   REGION FB Scanner
       #sScannerComm(iInit := "LBP_Chan1".A_Ref,
                     iReady := "DB_OPC_Laser".Scanner.In.Ready,
                     iStatus := "DB_OPC_Laser".Scanner.In.Status,
                     iStatusDescription := "DB_OPC_Laser".Scanner.In.StatusDescription,
                     iCheckNumber := "DB_OPC_Laser".Scanner.In.CheckNumber,
                     iPartOnFixture := "DB_PartManagement".sPosition.sFixture.Undrilled.Presence.Part OR "DB_PartManagement".sPosition.sFixture.Drilled.Presence.Part,
                     iStationNumber := #sScannerComm.iStationNumber,
                     iHoleNumber := #sScannerComm.iHoleNumber,
                     iJobListName := #sScannerComm.iJobListName,
                     iJobName := #sScannerComm.iJobName,
                     iMeasureZ := #sMeasureZ,
                     oEndOfJob => #sScannerComm.oEndOfJob,
                     ioRequestJob := "DB_OPC_Laser".Scanner.Out.RequestJob,
                     ioCheckNumber := "DB_OPC_Laser".Scanner.Out.CheckNumber,
                     oIsFirstJobOfPiece => "DB_OPC_Laser".Scanner.Out.Parameters.IsFirstJobOfPiece,
                     oStationNumber => "DB_OPC_Laser".Scanner.Out.Parameters.StationNumber,
                     oHoleNumber => "DB_OPC_Laser".Scanner.Out.Parameters.HoleNumber,
                     oJobListName => "DB_OPC_Laser".Scanner.Out.Parameters.JobListName,
                     oJobName => "DB_OPC_Laser".Scanner.Out.Parameters.JobName,
                     oMeasureZ => "DB_OPC_Laser".Scanner.Out.Parameters.MeasureZ,
                     oBadPart => #sScannerComm.oBadPart,
                     oGoodPart => #sScannerComm.oGoodPart,
                     ioRequestJob_NC := #sScannerComm.ioRequestJob_NC,
                     ioReady_NC := #sScannerComm.ioReady_NC);
   END_REGION

   REGION End of Job
       #sTimePulseWriteParam(IN := #sWriteR_ParamReq,
                             PT := T#100ms);
       IF #sTimePulseWriteParam.Q THEN
           #sWriteR_ParamReq := FALSE;
       END_IF;


       IF #sScannerComm.oEndOfJob THEN
           #sR96 := 0;
           #sR97 := 1;
           #sWriteR_ParamReq := TRUE;
       END_IF;

       IF #sWriteR_Param.Done THEN
           #sWriteR_ParamReq := FALSE;
       END_IF;
   END_REGION
END_FUNCTION_BLOCK

FUNCTION_BLOCK "FB_ScannerComm"   // FB85, SCL
{ S7_Optimized_Access := 'TRUE' }
// stored: MemoryReserve 100, SetENOAutomatically false
   VAR_INPUT
      iInit : Bool;
      iReady : Bool;   // From HMI OPC UA
      iStatus : DInt;   // From HMI OPC UA
      iStatusDescription : String;   // From HMI OPC UA
      iCheckNumber : Byte;   // From HMI OPC UA
      iPartOnFixture : Bool;
      iStationNumber : Byte;   // From NC ?
      iHoleNumber : DInt;   // From NC ?
      iJobListName : String;   // From NC ?
      iJobName : DInt;   // From NC ?
      iMeasureZ : LReal;   // From NC ?
   END_VAR
   VAR_OUTPUT
      oIsFirstJobOfPiece : Bool;
      oStationNumber : Byte;
      oHoleNumber : DInt;
      oJobListName : String;
      oJobName : String;
      oMeasureZ : LReal;
      oBadPart : Bool;
      oGoodPart : Bool;
      oEndOfJob : Bool;
   END_VAR
   VAR_IN_OUT
      ioRequestJob_NC : Bool;   // From NC ?
      ioReady_NC : Bool;   // From NC ?
      ioCheckNumber : Byte;
      ioRequestJob : Bool;
   END_VAR
   VAR
      sRT_PartOnFixture : R_TRIG;
      sRT_Ready { S7_SetPoint := 'True'} : R_TRIG;
      sEndOfJob { S7_SetPoint := 'True'} : Bool;
      sRT_RequestJob_NC : R_TRIG;
      sJobListName { S7_SetPoint := 'True'} : String;
      sJobName : String;
      sJobInProgress : Bool;
   END_VAR
BEGIN
   REGION Description header 
       //==================================================================================
       // POSALUX Swiss SA / (C) Copyright 2026
       //----------------------------------------------------------------------------------
       // Title: FB_ScannerComm
       // Comment/Function: 
       //
       // Author: Fabien WALDT
       // Engineering: TIA Portal v20
       //----------------------------------------------------------------------------------
       // Change log table:
       // Version  | Date     | Expert in charge | Changes applied
       // ---------|----------|------------------|------------------------------------
       // 00.00.01 | 20260330 | WFA              | First released version
       // ==================================================================================
   END_REGION

   REGION R_Trig
       #sRT_PartOnFixture(CLK := #iPartOnFixture);

       #sRT_Ready(CLK := #iReady);
       #sEndOfJob := #sRT_Ready.Q AND #sJobInProgress;

       #sRT_RequestJob_NC(CLK := #ioRequestJob_NC);
   END_REGION

   REGION Job
   #sJobListName := #iJobListName;
   #sJobName := DINT_TO_STRING(IN := #iJobName);

   IF #sJobName[1] = '+' THEN
       #sJobName := DELETE(IN := #sJobName, L := 1, P := 1);
   END_IF;
   END_REGION

   REGION Parameters
       // IsFirstJobOfPiece 
       IF #sRT_PartOnFixture.Q THEN
           #oIsFirstJobOfPiece := TRUE;
       ELSIF #sEndOfJob OR NOT #iPartOnFixture THEN
           #oIsFirstJobOfPiece := FALSE;
       END_IF;

       IF #sRT_RequestJob_NC.Q THEN
           // StationNumber 
           #oStationNumber := #iStationNumber;

           // HoleNumber 
           #oHoleNumber := #iHoleNumber;

           // JobListName 
           #oJobListName := #sJobListName;

           // JobName 
           #oJobName := #sJobName;

           // MeasureZ 
           #oMeasureZ := #iMeasureZ;

           // CheckNumber Increment
           #ioCheckNumber := #ioCheckNumber + 1;
           IF #ioCheckNumber > 255 OR #ioCheckNumber < 1 THEN
               #ioCheckNumber := 1;
           END_IF;

           // Reset Bad/Good Part
           #oBadPart := FALSE;
           #oGoodPart := FALSE;
       END_IF;
   END_REGION

   REGION Request Job
       IF #ioRequestJob_NC AND #iReady AND NOT #sJobInProgress THEN
           #sJobInProgress := TRUE;
           #ioRequestJob := TRUE;
       ELSIF (#ioRequestJob AND NOT #iReady) OR #iInit THEN
           #ioRequestJob := FALSE;
       END_IF;
   END_REGION

   REGION End of Job
       IF #sEndOfJob THEN
           IF #ioCheckNumber = #iCheckNumber AND #iStatus = 1 THEN
               #oGoodPart := TRUE;
           ELSE
               #oBadPart := TRUE;
           END_IF;
           #sJobInProgress := FALSE;
       END_IF;

       // Update Output
       #oEndOfJob := #sEndOfJob;
   END_REGION
END_FUNCTION_BLOCK

FUNCTION_BLOCK "FB_Part_Data"   // FB93, SCL
{ S7_Optimized_Access := 'TRUE' }
// stored: MemoryReserve 100, SetENOAutomatically false
   VAR
      Part_Data_Ident : "FB_ReadWrite_GUDs";
      sWriteDataEnable { S7_SetPoint := 'True'} : Bool;
      sNewPartDataIdent : Bool;
      RT_NewPartDataIdent : R_TRIG;
      sCurrentPartDataIdent { S7_SetPoint := 'True'} : String;
   END_VAR
   VAR_TEMP
      tIndex : Int;
   END_VAR
BEGIN
   REGION Description header 
       //==================================================================================
       // POSALUX Swiss SA / (C) Copyright 2026
       //----------------------------------------------------------------------------------
       // Title: FB_Part_Data
       // Comment/Function: 
       //
       // Author: Fabien WALDT
       // Engineering: TIA Portal v20
       //----------------------------------------------------------------------------------
       // Change log table:
       // Version  | Date     | Expert in charge | Changes applied
       // ---------|----------|------------------|------------------------------------
       // 00.00.01 | 20260518 | WFA              | First released version
       // ==================================================================================
   END_REGION

   REGION Data Init
       #Part_Data_Ident.sName := 'PART_DATA_IDENT';
       #Part_Data_Ident.sType := 4;
       #Part_Data_Ident.sNCK_channel := 1;
    //   #Part_Data_Ident.sWriteVal_String[0] := 'Test_ID_From_PLC';
   END_REGION

   REGION Call Read/Wrtite GUD
       #Part_Data_Ident();
   END_REGION

   REGION Convert DMC into String

   END_REGION

   REGION New Value
   // Convert DMC Array into String    
   Chars_TO_Strg(Chars:= "DB_DataPositions".Position[4].DMC,
                 pChars:= 0,
                 Cnt:= 19,
                 Strg=> #sCurrentPartDataIdent);

   // Check if new Part on Fixture
   IF #Part_Data_Ident.sWriteVal_String[0] <> #sCurrentPartDataIdent THEN
       #Part_Data_Ident.sWriteVal_String[0] := #sCurrentPartDataIdent;
       #sNewPartDataIdent := TRUE;
       END_IF;
   END_REGION

   // Il faut tout d'abord effectuer une lecture :
   // #Part_Data_Ident.sStart_rd
   // Pour obtenir #Part_Data_Ident.sRead_done
   // On peut alors effctuer une ecriture avec #Part_Data_Ident.sStart_wr
   // Pour obtenir #Part_Data_Ident.sWrite_done

   REGION Write Datas Request
       IF NOT #sWriteDataEnable THEN
           #Part_Data_Ident.sStart_rd := TRUE;
       END_IF;

   IF #Part_Data_Ident.sRead_done THEN
       #Part_Data_Ident.sStart_rd := FALSE;
       #sWriteDataEnable := TRUE;
   END_IF;

   #RT_NewPartDataIdent(CLK := #sNewPartDataIdent);
   IF #RT_NewPartDataIdent.Q AND #sWriteDataEnable THEN
       #Part_Data_Ident.sStart_wr := TRUE;
       #sNewPartDataIdent := FALSE;
   ELSIF #Part_Data_Ident.sWrite_done THEN
       #Part_Data_Ident.sStart_wr := FALSE;
   END_IF;
   END_REGION
END_FUNCTION_BLOCK

FUNCTION_BLOCK "FB_ReadWrite_GUDs"   // FB1200, SCL
{ S7_Optimized_Access := 'TRUE' }
// stored: AutoNumber false, MemoryReserve 100, SetENOAutomatically false
   VAR
      sStart_rd { ExternalAccessible := 'False'; ExternalVisible := 'False'; ExternalWritable := 'False'} : Bool;
      sNCK_channel { ExternalAccessible := 'False'; ExternalVisible := 'False'; ExternalWritable := 'False'} : Byte;   // 0:GUD NCK, 1:GUD Chan1, 2:GUD Chan2 etc...
      sType { ExternalAccessible := 'False'; ExternalVisible := 'False'; ExternalWritable := 'False'} : Int;   // 0:Bool, 1:Int, 2:DWord, 3:Real, 4:String
      sName { ExternalAccessible := 'False'; ExternalVisible := 'False'; ExternalWritable := 'False'} : String;   // GUD Name
      sIndex1 { ExternalAccessible := 'False'; ExternalVisible := 'False'; ExternalWritable := 'False'} : Int;
      sindex2 { ExternalAccessible := 'False'; ExternalVisible := 'False'; ExternalWritable := 'False'} : Int;
      sToken_GUD { ExternalAccessible := 'False'; ExternalVisible := 'False'; ExternalWritable := 'False'} : "UDT_Token_GUD";
      sValue_bit { ExternalAccessible := 'False'; ExternalVisible := 'False'; ExternalWritable := 'False'} : Bool;
      sValue_int { ExternalAccessible := 'False'; ExternalVisible := 'False'; ExternalWritable := 'False'} : Int;
      sValue_double { ExternalAccessible := 'False'; ExternalVisible := 'False'; ExternalWritable := 'False'} : DWord;
      sValue_real { ExternalAccessible := 'False'; ExternalVisible := 'False'; ExternalWritable := 'False'} : Real;
      sValue_String { ExternalAccessible := 'False'; ExternalVisible := 'False'; ExternalWritable := 'False'} : String;
      sStatus_rd { ExternalAccessible := 'False'; ExternalVisible := 'False'; ExternalWritable := 'False'} : Word;
      sRead_done { ExternalAccessible := 'False'; ExternalVisible := 'False'; ExternalWritable := 'False'} : Bool;
      sRead_done_Mem { ExternalAccessible := 'False'; ExternalVisible := 'False'; ExternalWritable := 'False'} : Bool;
      sStart_wr { ExternalAccessible := 'False'; ExternalVisible := 'False'; ExternalWritable := 'False'} : Bool;
      sNumVar_wr { ExternalAccessible := 'False'; ExternalVisible := 'False'; ExternalWritable := 'False'} : Int := 1;
      sAddr_wr { ExternalAccessible := 'False'; ExternalVisible := 'False'; ExternalWritable := 'False'} : Array[0..7] of "UDT_Token_GUD";
      sColumn_wr { ExternalAccessible := 'False'; ExternalVisible := 'False'; ExternalWritable := 'False'} : Array[0..7] of Word;
      sLine_wr { ExternalAccessible := 'False'; ExternalVisible := 'False'; ExternalWritable := 'False'} : Array[0..7] of Word;
      sStatus_wr { ExternalAccessible := 'False'; ExternalVisible := 'False'; ExternalWritable := 'False'} : Word;
      sWrite_done { ExternalAccessible := 'False'; ExternalVisible := 'False'; ExternalWritable := 'False'} : Bool;
      sWriteVal_bit { ExternalAccessible := 'False'; ExternalVisible := 'False'; ExternalWritable := 'False'} : Array[0..7] of Bool;
      sWriteVal_int { ExternalAccessible := 'False'; ExternalVisible := 'False'; ExternalWritable := 'False'} : Array[0..7] of Int;
      sWriteVal_double { ExternalAccessible := 'False'; ExternalVisible := 'False'; ExternalWritable := 'False'} : Array[0..7] of DWord;
      sWriteVal_Real { ExternalAccessible := 'False'; ExternalVisible := 'False'; ExternalWritable := 'False'} : Array[0..7] of DWord;
      sWriteVal_String { ExternalAccessible := 'False'; ExternalVisible := 'False'; ExternalWritable := 'False'} : Array[0..7] of String;
      sLBP_ReadGUD_Instance { ExternalAccessible := 'False'; ExternalVisible := 'False'; ExternalWritable := 'False'} : "LBP_ReadGUD";
      sLBP_WriteGUD_Instance { ExternalAccessible := 'False'; ExternalVisible := 'False'; ExternalWritable := 'False'} : "LBP_WriteVar";
   END_VAR
   VAR_TEMP
      tArea : Byte;
      tUnit : Byte;
      tError : Bool;
      tStatus : Word;
      tLoop_I : Int;
   END_VAR
   // sColumn_wr[0..7] := 16#1;
   // sLine_wr[0..7] := 16#1;
BEGIN
   REGION Reading
       IF #sNCK_channel = 0 THEN
           #tArea := 0;
           #tUnit := 1;
       ELSE
           #tArea := 2;
           #tUnit := #sNCK_channel;
       END_IF;

       CASE #sType OF
           0:
               #sLBP_ReadGUD_Instance(Req := #sStart_rd,
                                     Addr := #sName,
                                     Area := #tArea,
                                     Unit := #tUnit,
                                     Index1 := #sIndex1,
                                     Index2 := #sindex2,
                                     CnvtToken := TRUE,
                                     VarToken := #sToken_GUD,
                                     Error => #tError,
                                     Done => #sRead_done,
                                     State => #tStatus,
                                     RD := #sValue_bit);
           1:
               #sLBP_ReadGUD_Instance(Req := #sStart_rd,
                                     Addr := #sName,
                                     Area := #tArea,
                                     Unit := #tUnit,
                                     Index1 := #sIndex1,
                                     Index2 := #sindex2,
                                     CnvtToken := TRUE,
                                     VarToken := #sToken_GUD,
                                     Error => #tError,
                                     Done => #sRead_done,
                                     State => #tStatus,
                                     RD := #sValue_int);

           2:
               #sLBP_ReadGUD_Instance(Req := #sStart_rd,
                                     Addr := #sName,
                                     Area := #tArea,
                                     Unit := #tUnit,
                                     Index1 := #sIndex1,
                                     Index2 := #sindex2,
                                     CnvtToken := TRUE,
                                     VarToken := #sToken_GUD,
                                     Error => #tError,
                                     Done => #sRead_done,
                                     State => #tStatus,
                                     RD := #sValue_double);

           3:
               #sLBP_ReadGUD_Instance(Req := #sStart_rd,
                                     Addr := #sName,
                                     Area := #tArea,
                                     Unit := #tUnit,
                                     Index1 := #sIndex1,
                                     Index2 := #sindex2,
                                     CnvtToken := TRUE,
                                     VarToken := #sToken_GUD,
                                     Error => #tError,
                                     Done => #sRead_done,
                                     State => #tStatus,
                                     RD := #sValue_real);

           4:
               #sLBP_ReadGUD_Instance(Req := #sStart_rd,
                                     Addr := #sName,
                                     Area := #tArea,
                                     Unit := #tUnit,
                                     Index1 := #sIndex1,
                                     Index2 := #sindex2,
                                     CnvtToken := TRUE,
                                     VarToken := #sToken_GUD,
                                     Error => #tError,
                                     Done => #sRead_done,
                                     State => #tStatus,
                                     RD := #sValue_String);


       END_CASE;

       IF #sRead_done OR #tError THEN
           #sRead_done := TRUE;
           #sStatus_rd := #tStatus;
           #sStart_rd := FALSE;
       END_IF;
       IF #sRead_done AND NOT #sRead_done_Mem THEN
           FOR #tLoop_I := 1 TO 8 DO
               IF #tLoop_I <= #sNumVar_wr THEN
                 #sAddr_wr[#tLoop_I - 1] := #sToken_GUD;
               END_IF;
           END_FOR;
           #sRead_done_Mem := TRUE;
       END_IF;

   END_REGION


   REGION Writing

       CASE #sType OF
           0:
               #sLBP_WriteGUD_Instance(Req := #sStart_wr AND #sRead_done_Mem,
                                      NumVar := #sNumVar_wr,
                                      Addr1 := #sAddr_wr[0],
                                      Line1 := #sLine_wr[0],
                                      Column1 := #sColumn_wr[0],
                                      Addr2 := #sAddr_wr[1],
                                      Line2 := #sLine_wr[1],
                                      Column2 := #sColumn_wr[1],
                                      Addr3 := #sAddr_wr[2],
                                      Line3 := #sLine_wr[2],
                                      Column3 := #sColumn_wr[2],
                                      Addr4 := #sAddr_wr[3],
                                      Line4 := #sLine_wr[3],
                                      Column4 := #sColumn_wr[3],
                                      Addr5 := #sAddr_wr[4],
                                      Line5 := #sLine_wr[4],
                                      Column5 := #sColumn_wr[4],
                                      Addr6 := #sAddr_wr[5],
                                      Line6 := #sLine_wr[5],
                                      Column6 := #sColumn_wr[5],
                                      Addr7 := #sAddr_wr[6],
                                      Line7 := #sLine_wr[6],
                                      Column7 := #sColumn_wr[6],
                                      Addr8 := #sAddr_wr[7],
                                      Line8 := #sLine_wr[7],
                                      Column8 := #sColumn_wr[7],
                                      Error => #tError,
                                      Done => #sWrite_done,
                                      State => #tStatus,
                                      SD1 := #sWriteVal_bit[0],
                                      SD2 := #sWriteVal_bit[1],
                                      SD3 := #sWriteVal_bit[2],
                                      SD4 := #sWriteVal_bit[3],
                                      SD5 := #sWriteVal_bit[4],
                                      SD6 := #sWriteVal_bit[5],
                                      SD7 := #sWriteVal_bit[6],
                                      SD8 := #sWriteVal_bit[7]);
           1:
               #sLBP_WriteGUD_Instance(Req := #sStart_wr AND #sRead_done_Mem,
                                      NumVar := #sNumVar_wr,
                                      Addr1 := #sAddr_wr[0],
                                      Line1 := #sLine_wr[0],
                                      Column1 := #sColumn_wr[0],
                                      Addr2 := #sAddr_wr[1],
                                      Line2 := #sLine_wr[1],
                                      Column2 := #sColumn_wr[1],
                                      Addr3 := #sAddr_wr[2],
                                      Line3 := #sLine_wr[2],
                                      Column3 := #sColumn_wr[2],
                                      Addr4 := #sAddr_wr[3],
                                      Line4 := #sLine_wr[3],
                                      Column4 := #sColumn_wr[3],
                                      Addr5 := #sAddr_wr[4],
                                      Line5 := #sLine_wr[4],
                                      Column5 := #sColumn_wr[4],
                                      Addr6 := #sAddr_wr[5],
                                      Line6 := #sLine_wr[5],
                                      Column6 := #sColumn_wr[5],
                                      Addr7 := #sAddr_wr[6],
                                      Line7 := #sLine_wr[6],
                                      Column7 := #sColumn_wr[6],
                                      Addr8 := #sAddr_wr[7],
                                      Line8 := #sLine_wr[7],
                                      Column8 := #sColumn_wr[7],
                                      Error => #tError,
                                      Done => #sWrite_done,
                                      State => #tStatus,
                                      SD1 := #sWriteVal_int[0],
                                      SD2 := #sWriteVal_int[1],
                                      SD3 := #sWriteVal_int[2],
                                      SD4 := #sWriteVal_int[3],
                                      SD5 := #sWriteVal_int[4],
                                      SD6 := #sWriteVal_int[5],
                                      SD7 := #sWriteVal_int[6],
                                      SD8 := #sWriteVal_int[7]);

           2:
               #sLBP_WriteGUD_Instance(Req := #sStart_wr AND #sRead_done_Mem,
                                      NumVar := #sNumVar_wr,
                                      Addr1 := #sAddr_wr[0],
                                      Line1 := #sLine_wr[0],
                                      Column1 := #sColumn_wr[0],
                                      Addr2 := #sAddr_wr[1],
                                      Line2 := #sLine_wr[1],
                                      Column2 := #sColumn_wr[1],
                                      Addr3 := #sAddr_wr[2],
                                      Line3 := #sLine_wr[2],
                                      Column3 := #sColumn_wr[2],
                                      Addr4 := #sAddr_wr[3],
                                      Line4 := #sLine_wr[3],
                                      Column4 := #sColumn_wr[3],
                                      Addr5 := #sAddr_wr[4],
                                      Line5 := #sLine_wr[4],
                                      Column5 := #sColumn_wr[4],
                                      Addr6 := #sAddr_wr[5],
                                      Line6 := #sLine_wr[5],
                                      Column6 := #sColumn_wr[5],
                                      Addr7 := #sAddr_wr[6],
                                      Line7 := #sLine_wr[6],
                                      Column7 := #sColumn_wr[6],
                                      Addr8 := #sAddr_wr[7],
                                      Line8 := #sLine_wr[7],
                                      Column8 := #sColumn_wr[7],
                                      Error => #tError,
                                      Done => #sWrite_done,
                                      State => #tStatus,
                                      SD1 := #sWriteVal_double[0],
                                      SD2 := #sWriteVal_double[1],
                                      SD3 := #sWriteVal_double[2],
                                      SD4 := #sWriteVal_double[3],
                                      SD5 := #sWriteVal_double[4],
                                      SD6 := #sWriteVal_double[5],
                                      SD7 := #sWriteVal_double[6],
                                      SD8 := #sWriteVal_double[7]);

           3:
               #sLBP_WriteGUD_Instance(Req := #sStart_wr AND #sRead_done_Mem,
                                      NumVar := #sNumVar_wr,
                                      Addr1 := #sAddr_wr[0],
                                      Line1 := #sLine_wr[0],
                                      Column1 := #sColumn_wr[0],
                                      Addr2 := #sAddr_wr[1],
                                      Line2 := #sLine_wr[1],
                                      Column2 := #sColumn_wr[1],
                                      Addr3 := #sAddr_wr[2],
                                      Line3 := #sLine_wr[2],
                                      Column3 := #sColumn_wr[2],
                                      Addr4 := #sAddr_wr[3],
                                      Line4 := #sLine_wr[3],
                                      Column4 := #sColumn_wr[3],
                                      Addr5 := #sAddr_wr[4],
                                      Line5 := #sLine_wr[4],
                                      Column5 := #sColumn_wr[4],
                                      Addr6 := #sAddr_wr[5],
                                      Line6 := #sLine_wr[5],
                                      Column6 := #sColumn_wr[5],
                                      Addr7 := #sAddr_wr[6],
                                      Line7 := #sLine_wr[6],
                                      Column7 := #sColumn_wr[6],
                                      Addr8 := #sAddr_wr[7],
                                      Line8 := #sLine_wr[7],
                                      Column8 := #sColumn_wr[7],
                                      Error => #tError,
                                      Done => #sWrite_done,
                                      State => #tStatus,
                                      SD1 := #sWriteVal_Real[0],
                                      SD2 := #sWriteVal_Real[1],
                                      SD3 := #sWriteVal_Real[2],
                                      SD4 := #sWriteVal_Real[3],
                                      SD5 := #sWriteVal_Real[4],
                                      SD6 := #sWriteVal_Real[5],
                                      SD7 := #sWriteVal_Real[6],
                                      SD8 := #sWriteVal_Real[7]);

           4:
               #sLBP_WriteGUD_Instance(Req := #sStart_wr AND #sRead_done_Mem,
                                      NumVar := #sNumVar_wr,
                                      Addr1 := #sAddr_wr[0],
                                      Line1 := #sLine_wr[0],
                                      Column1 := #sColumn_wr[0],
                                      Addr2 := #sAddr_wr[1],
                                      Line2 := #sLine_wr[1],
                                      Column2 := #sColumn_wr[1],
                                      Addr3 := #sAddr_wr[2],
                                      Line3 := #sLine_wr[2],
                                      Column3 := #sColumn_wr[2],
                                      Addr4 := #sAddr_wr[3],
                                      Line4 := #sLine_wr[3],
                                      Column4 := #sColumn_wr[3],
                                      Addr5 := #sAddr_wr[4],
                                      Line5 := #sLine_wr[4],
                                      Column5 := #sColumn_wr[4],
                                      Addr6 := #sAddr_wr[5],
                                      Line6 := #sLine_wr[5],
                                      Column6 := #sColumn_wr[5],
                                      Addr7 := #sAddr_wr[6],
                                      Line7 := #sLine_wr[6],
                                      Column7 := #sColumn_wr[6],
                                      Addr8 := #sAddr_wr[7],
                                      Line8 := #sLine_wr[7],
                                      Column8 := #sColumn_wr[7],
                                      Error => #tError,
                                      Done => #sWrite_done,
                                      State => #tStatus,
                                      SD1 := #sWriteVal_String[0],
                                      SD2 := #sWriteVal_String[1],
                                      SD3 := #sWriteVal_String[2],
                                      SD4 := #sWriteVal_String[3],
                                      SD5 := #sWriteVal_String[4],
                                      SD6 := #sWriteVal_String[5],
                                      SD7 := #sWriteVal_String[6],
                                      SD8 := #sWriteVal_String[7]);
       END_CASE;

       IF #sWrite_done OR #tError THEN
           #sWrite_done := TRUE;
           #sStatus_wr := #tStatus;
           #sStart_wr := FALSE;
       END_IF;


   END_REGION
END_FUNCTION_BLOCK

FUNCTION_BLOCK "FB_Recipe"   // FB81, SCL
{ S7_Optimized_Access := 'TRUE' }
// stored: AutoNumber false, MemoryReserve 100, SetENOAutomatically false
BEGIN
   REGION Description header 
       //==================================================================================
       // POSALUX Swiss SA / (C) Copyright 2026
       //----------------------------------------------------------------------------------
       // Title: FB_Recipe
       // Comment/Function: 
       //
       // Author: Fabien WALDT
       // Engineering: TIA Portal v20
       //----------------------------------------------------------------------------------
       // Change log table:
       // Version  | Date     | Expert in charge | Changes applied
       // ---------|----------|------------------|------------------------------------
       // 00.00.01 | 20260427 | WFA              | First released version
       // ==================================================================================
   END_REGION

   REGION Current
       "DB_OPC_Recipe".Current.RecipeId := "DB_OPC_Recipe".Current.RecipeId;
       "DB_OPC_Recipe".Current.RecipeVersionGuid := "DB_OPC_Recipe".Current.RecipeVersionGuid;
   END_REGION

   REGION Data
       "DB_OPC_Recipe".Data.LaserJobListName := "DB_OPC_Recipe".Data.LaserJobListName;
       "DB_OPC_Recipe".Data.RecipeId := "DB_OPC_Recipe".Data.RecipeId;
       "DB_OPC_Recipe".Data.RecipeName := "DB_OPC_Recipe".Data.RecipeName;
       "DB_OPC_Recipe".Data.RecipeVersionGuid := "DB_OPC_Recipe".Data.RecipeVersionGuid;

       // Station 1
       // General \ Detections \ WorkPart
       "DB_OPC_Recipe".Data.Station1.General.Detections.WorkPart.Max := "DB_OPC_Recipe".Data.Station1.General.Detections.WorkPart.Max;
       "DB_OPC_Recipe".Data.Station1.General.Detections.WorkPart.Min := "DB_OPC_Recipe".Data.Station1.General.Detections.WorkPart.Min;
       // General \ GasPressure
        "DB_OPC_Recipe".Data.Station1.General.GazPressure.WorkLaserDefault := "DB_OPC_Recipe".Data.Station1.General.GazPressure.WorkLaserDefault;
   END_REGION

   REGION TransfertToPlc
       IF "DB_OPC_Recipe".TransferToPlc THEN
           "DB_OPC_Recipe".Current.RecipeId := "DB_OPC_Recipe".Data.RecipeId;
           "DB_OPC_Recipe".Current.RecipeVersionGuid := "DB_OPC_Recipe".Data.RecipeVersionGuid;
           "DB_Scanner".sScannerComm.iJobListName := "DB_OPC_Recipe".Data.LaserJobListName;
       //    "DB_HMISetting".GasAssistSetPoint := LREAL_TO_REAL("DB_OPC_Recipe".Data.Station1.General.GazPressure.WorkLaserDefault);   WAF A LIBERER QUAND RECETTE OK
       //    "DB_GestionFixture".sFixturePartControl.iProdOK_LimHigh := LREAL_TO_REAL("DB_OPC_Recipe".Data.Station1.General.Detections.WorkPart.Max);  WAF A LIBERER QUAND RECETTE OK
       //    "DB_GestionFixture".sFixturePartControl.iProdOK_LimLow := LREAL_TO_REAL("DB_OPC_Recipe".Data.Station1.General.Detections.WorkPart.Min);   WAF A LIBERER QUAND RECETTE OK
           "DB_OPC_Recipe".TransferToPlc := FALSE;
       END_IF;
   END_REGION
END_FUNCTION_BLOCK

FUNCTION_BLOCK "FB_PartManagement"   // FB86, SCL
{ S7_Optimized_Access := 'TRUE' }
// stored: MemoryReserve 100, SetENOAutomatically false
   VAR
      sShuttle1DrilledPart : "FB_StatusPart";
      sShuttle1UndrilledPart { S7_SetPoint := 'True'} : "FB_StatusPart";
      sShuttle2DrilledPart { S7_SetPoint := 'True'} : "FB_StatusPart";
      sShuttle2UndrilledPart { S7_SetPoint := 'True'} : "FB_StatusPart";
      sShuttle1DrilledBw : "FB_StatusPart";
      sShuttle1UndrilledBw { S7_SetPoint := 'True'} : "FB_StatusPart";
      sShuttle2DrilledBw { S7_SetPoint := 'True'} : "FB_StatusPart";
      sShuttle2UndrilledBw { S7_SetPoint := 'True'} : "FB_StatusPart";
      sGripperDrilledPart : "FB_StatusPart";
      sGripperUndrilledPart { S7_SetPoint := 'True'} : "FB_StatusPart";
      sGripperDrilledBw : "FB_StatusPart";
      sGripperUndrilledBw { S7_SetPoint := 'True'} : "FB_StatusPart";
      sFixtureDrilledPart : "FB_StatusPart";
      sFixtureUndrilledPart { S7_SetPoint := 'True'} : "FB_StatusPart";
      sFixtureDrilledBw : "FB_StatusPart";
      sFixtureUndrilledBw { S7_SetPoint := 'True'} : "FB_StatusPart";
      sPosition { S7_SetPoint := 'True'} : "FB_Position";
   END_VAR
BEGIN
   REGION Description header 
       //==================================================================================
       // POSALUX Swiss SA / (C) Copyright 2026
       //----------------------------------------------------------------------------------
       // Title: FB_PartManagement
       // Comment/Function: 
       //
       // Author: Fabien WALDT
       // Engineering: TIA Portal v20
       //----------------------------------------------------------------------------------
       // Change log table:
       // Version  | Date     | Expert in charge | Changes applied
       // ---------|----------|------------------|------------------------------------
       // 00.00.01 | 20260310 | WFA              | First released version
       // ==================================================================================
   END_REGION

   REGION Shuttle 1 States
       // Drilled Part
       #sShuttle1DrilledPart(iGood := #sPosition.sShuttle1.Drilled.Presence.Part AND NOT #sShuttle1DrilledPart.iBad,
                             iUnknown := #sShuttle1DrilledPart.iUnknown,
                             iBad := #sShuttle1DrilledPart.iBad,
                             iAbsent := NOT #sPosition.sShuttle1.Drilled.Presence.Part,
                             iPresentUnexpected := "DB_LoaderShuttle1".sControlIn.sExtraPartCtrlDrilled OR "DB_LoaderShuttle1".sControlOut.sExtraPartCtrlDrilled,
                             iAbsentUnexpected := "DB_LoaderShuttle1".sControlIn.sMissingPartCtrlDrilled OR "DB_LoaderShuttle1".sControlOut.sMissingPartCtrlDrilled,
                             oStatus => #sPosition.sShuttle1.Drilled.States.Part);

       // Undrilled Part
       #sShuttle1UndrilledPart(iGood := #sPosition.sShuttle1.Undrilled.Presence.Part AND NOT #sShuttle1UndrilledPart.iBad,
                               iUnknown := #sShuttle1UndrilledPart.iUnknown,
                               iBad := #sShuttle1UndrilledPart.iBad,
                               iAbsent := NOT #sPosition.sShuttle1.Undrilled.Presence.Part,
                               iPresentUnexpected := "DB_LoaderShuttle1".sControlIn.sExtraPartCtrlUndrilled OR "DB_LoaderShuttle1".sControlOut.sExtraPartCtrlUndrilled,
                               iAbsentUnexpected := "DB_LoaderShuttle1".sControlIn.sMissingPartCtrlUndrilled OR "DB_LoaderShuttle1".sControlOut.sMissingPartCtrlUndrilled,
                               oStatus => #sPosition.sShuttle1.Undrilled.States.Part);
       // Drilled Bw
       #sShuttle1DrilledBw(iGood := #sPosition.sShuttle1.Drilled.Presence.BW AND NOT #sShuttle1DrilledBw.iBad,
                           iUnknown := #sShuttle1DrilledBw.iUnknown,
                           iBad := #sShuttle1DrilledBw.iBad,
                           iAbsent := NOT #sPosition.sShuttle1.Drilled.Presence.BW,
                           iPresentUnexpected := FALSE,
                           iAbsentUnexpected := FALSE,
                           oStatus => #sPosition.sShuttle1.Drilled.States.BW);

       // Undrilled Bw
       #sShuttle1UndrilledBw(iGood := #sPosition.sShuttle1.Undrilled.Presence.BW AND NOT #sShuttle1UndrilledBw.iBad,
                             iUnknown := #sShuttle1UndrilledBw.iUnknown,
                             iBad := #sShuttle1UndrilledBw.iBad,
                             iAbsent := NOT #sPosition.sShuttle1.Undrilled.Presence.BW,
                             iPresentUnexpected := "DB_LoaderShuttle1".sBwControlIn.sExtraBwCtrl,
                             iAbsentUnexpected := "DB_LoaderShuttle1".sBwControlIn.sMissingBwCtrl,
                             oStatus => #sPosition.sShuttle1.Undrilled.States.BW);
   END_REGION

   REGION Shuttle 2 States
       // Drilled Part
       #sShuttle2DrilledPart(iGood := #sPosition.sShuttle2.Drilled.Presence.Part AND NOT #sShuttle2DrilledPart.iBad,
                             iUnknown := #sShuttle2DrilledPart.iUnknown,
                             iBad := #sShuttle2DrilledPart.iBad,
                             iAbsent := NOT #sPosition.sShuttle2.Drilled.Presence.Part,
                             iPresentUnexpected := "DB_LoaderShuttle2".sControlIn.sExtraPartCtrlDrilled OR "DB_LoaderShuttle2".sControlOut.sExtraPartCtrlDrilled,
                             iAbsentUnexpected := "DB_LoaderShuttle2".sControlIn.sMissingPartCtrlDrilled OR "DB_LoaderShuttle2".sControlOut.sMissingPartCtrlDrilled,
                             oStatus => #sPosition.sShuttle2.Drilled.States.Part);

       // Undrilled Part
       #sShuttle2UndrilledPart(iGood := #sPosition.sShuttle2.Undrilled.Presence.Part AND NOT #sShuttle2UndrilledPart.iBad,
                               iUnknown := #sShuttle2UndrilledPart.iUnknown,
                               iBad := #sShuttle2UndrilledPart.iBad,
                               iAbsent := NOT #sPosition.sShuttle2.Undrilled.Presence.Part,
                               iPresentUnexpected := "DB_LoaderShuttle2".sControlIn.sExtraPartCtrlUndrilled OR "DB_LoaderShuttle2".sControlOut.sExtraPartCtrlUndrilled,
                               iAbsentUnexpected := "DB_LoaderShuttle2".sControlIn.sMissingPartCtrlUndrilled OR "DB_LoaderShuttle2".sControlOut.sMissingPartCtrlUndrilled,
                               oStatus => #sPosition.sShuttle2.Undrilled.States.Part);
       // Drilled Bw
       #sShuttle2DrilledBw(iGood := #sPosition.sShuttle2.Drilled.Presence.BW AND NOT #sShuttle2DrilledBw.iBad,
                           iUnknown := #sShuttle2DrilledBw.iUnknown,
                           iBad := #sShuttle2DrilledBw.iBad,
                           iAbsent := NOT #sPosition.sShuttle2.Drilled.Presence.BW,
                           iPresentUnexpected := FALSE,
                           iAbsentUnexpected := FALSE,
                           oStatus => #sPosition.sShuttle2.Drilled.States.BW);

       // Undrilled Bw
       #sShuttle2UndrilledBw(iGood := #sPosition.sShuttle2.Undrilled.Presence.BW AND NOT #sShuttle2UndrilledBw.iBad,
                             iUnknown := #sShuttle2UndrilledBw.iUnknown,
                             iBad := #sShuttle2UndrilledBw.iBad,
                             iAbsent := NOT #sPosition.sShuttle2.Undrilled.Presence.BW,
                             iPresentUnexpected := "DB_LoaderShuttle2".sBwControlIn.sExtraBwCtrl,
                             iAbsentUnexpected := "DB_LoaderShuttle2".sBwControlIn.sMissingBwCtrl,
                             oStatus => #sPosition.sShuttle2.Undrilled.States.BW);
   END_REGION

   REGION Gripper States
       // Drilled Part
       #sGripperDrilledPart(iGood := #sPosition.sGripper.Drilled.Presence.Part AND NOT #sGripperDrilledPart.iBad,
                            iUnknown := #sGripperDrilledPart.iUnknown,
                            iBad := #sGripperDrilledPart.iBad,
                            iAbsent := NOT #sPosition.sGripper.Drilled.Presence.Part,
                            iPresentUnexpected := "DB_ExtraMissingPart".sExtraPartDrilledGripper,
                            iAbsentUnexpected := "DB_ExtraMissingPart".sMissingPartDrilledGripper,
                            oStatus => #sPosition.sGripper.Drilled.States.Part);

       // Undrilled Part
       #sGripperUndrilledPart(iGood := #sPosition.sGripper.Undrilled.Presence.Part AND NOT #sGripperUndrilledPart.iBad,
                              iUnknown := #sGripperUndrilledPart.iUnknown,
                              iBad := #sGripperUndrilledPart.iBad,
                              iAbsent := NOT #sPosition.sGripper.Undrilled.Presence.Part,
                              iPresentUnexpected := "DB_ExtraMissingPart".sExtraPartUndrilledGripper,
                              iAbsentUnexpected := "DB_ExtraMissingPart".sMissingPartUndrilledGripper,
                              oStatus => #sPosition.sGripper.Undrilled.States.Part);
       // Drilled Bw
       #sGripperDrilledBw(iGood := #sPosition.sGripper.Drilled.Presence.BW AND NOT #sGripperDrilledBw.iBad,
                          iUnknown := #sGripperDrilledBw.iUnknown,
                          iBad := #sGripperDrilledBw.iBad,
                          iAbsent := NOT #sPosition.sGripper.Drilled.Presence.BW,
                          iPresentUnexpected := "DB_ExtraMissingPart".sExtraPartDrilledGripper,
                          iAbsentUnexpected := "DB_ExtraMissingPart".sMissingPartDrilledGripper,
                          oStatus => #sPosition.sGripper.Drilled.States.BW);

       // Undrilled Bw
       #sGripperUndrilledBw(iGood := #sPosition.sGripper.Undrilled.Presence.BW AND NOT #sGripperUndrilledBw.iBad,
                            iUnknown := #sGripperUndrilledBw.iUnknown,
                            iBad := #sGripperUndrilledBw.iBad,
                            iAbsent := NOT #sPosition.sGripper.Undrilled.Presence.BW,
                            iPresentUnexpected := "DB_ExtraMissingPart".sExtraPartUndrilledGripper,
                            iAbsentUnexpected := "DB_ExtraMissingPart".sMissingPartUndrilledGripper,
                            oStatus => #sPosition.sGripper.Undrilled.States.BW);
   END_REGION

   REGION Fixture States
       // Drilled - Part
       #sFixtureDrilledPart(iGood := #sPosition.sFixture.Drilled.Presence.Part AND NOT #sFixtureDrilledPart.iBad,
                            iUnknown := #sFixtureDrilledPart.iUnknown,
                            iBad := "DB_ScannerComm".oBadPart,
                            iAbsent := NOT #sPosition.sFixture.Drilled.Presence.Part AND NOT #sPosition.sFixture.Undrilled.Presence.Part,
                            iPresentUnexpected := "DB_ExtraMissingPart".sExtraPartFixture,
                            iAbsentUnexpected := "DB_ExtraMissingPart".sMissingPartFixture,
                            oStatus => #sPosition.sFixture.Drilled.States.Part);

        // Undrilled Part
       #sFixtureUndrilledPart(iGood := #sPosition.sFixture.Undrilled.Presence.Part,
                              iUnknown := #sFixtureUndrilledPart.iUnknown,
                              iBad := #sFixtureUndrilledPart.iBad,
                              iAbsent := NOT #sPosition.sFixture.Undrilled.Presence.Part,
                              iPresentUnexpected := "DB_ExtraMissingPart".sExtraPartFixture,
                              iAbsentUnexpected := "DB_ExtraMissingPart".sMissingPartFixture,
                              oStatus => #sPosition.sFixture.Undrilled.States.Part);
       // Drilled Bw 
         #sFixtureDrilledBw(iGood := (#sPosition.sFixture.Drilled.Presence.BW OR #sPosition.sFixture.Undrilled.Presence.BW) AND NOT #sGripperDrilledBw.iBad,
                            iUnknown := #sFixtureDrilledBw.iUnknown,
                            iBad := #sFixtureDrilledBw.iBad,
                            iAbsent := NOT #sPosition.sFixture.Drilled.Presence.BW AND NOT #sPosition.sFixture.Undrilled.Presence.BW,
                            iPresentUnexpected := "DB_ExtraMissingPart".sExtraPartFixture,
                            iAbsentUnexpected := "DB_ExtraMissingPart".sMissingPartFixture,
                            oStatus => #sPosition.sFixture.Drilled.States.BW);

       // Undrilled Bw
       #sGripperUndrilledBw(iGood := #sPosition.sFixture.Undrilled.Presence.BW,
                            iUnknown := #sGripperUndrilledBw.iUnknown,
                            iBad := #sGripperUndrilledBw.iBad,
                            iAbsent := NOT #sPosition.sFixture.Undrilled.Presence.BW,
                            iPresentUnexpected := "DB_ExtraMissingPart".sExtraPartFixture,
                            iAbsentUnexpected := "DB_ExtraMissingPart".sMissingPartFixture,
                            oStatus => #sPosition.sFixture.Undrilled.States.BW);
   END_REGION

   REGION Position
       #sPosition(iCondPartInSh1 := (("DB_LoaderShuttle1".sExtLoadUnload.sCurrent_Step_NB = 60 OR "DB_LoaderShuttle1".sExtLoadUnload.sCurrent_Step_NB = 120) AND NOT "DB_WorkingModes".sEmptying),
                  iCondBwInSh1 := "DB_LoaderShuttle1".sBwLoadUnload.sInterface.JobDone AND "DB_LoaderShuttle1".sBwLoadUnload.iLoadReq,
                  iCondPartInSh2 := (("DB_LoaderShuttle2".sExtLoadUnload.sCurrent_Step_NB = 60 OR "DB_LoaderShuttle2".sExtLoadUnload.sCurrent_Step_NB = 120) AND NOT "DB_WorkingModes".sEmptying),
                  iCondBwInSh2 := "DB_LoaderShuttle2".sBwLoadUnload.sInterface.JobDone AND "DB_LoaderShuttle2".sBwLoadUnload.iLoadReq,
                  iCondPartPresCtrlInSh1 := "DB_LoaderShuttle1".sControlIn.sCurrent_Step_NB = 140 AND NOT "DB_WorkingModes".sEmptying,
                  iCondBWPresCtrlInSh1 := "DB_LoaderShuttle1".sBwControlIn.sCurrent_Step_NB = 40,
                  iCondPartPresCtrlInSh2 := "DB_LoaderShuttle2".sControlIn.sCurrent_Step_NB = 140,
                  iCondBWPresCtrlInSh2 := "DB_LoaderShuttle2".sBwControlIn.sCurrent_Step_NB = 40,
                  iCondPartPresCtrlOutSh1 := "DB_LoaderShuttle1".sControlOut.sCurrent_Step_NB = 140,
                  iCondPartPresCtrlOutSh2 := "DB_LoaderShuttle2".sControlOut.sCurrent_Step_NB = 140,
                  iUndrilledPartPresence := "DB_DigitalInputsBW_Station".sUndrilledPartCtrl.sSWStatus,
                  iDrilledPartPresence := "DB_DigitalInputsBW_Station".sDrilledPartCtrl.sSWStatus,
                  iUndrilledBWPresence := "DB_DigitalInputsBW_Station".sBwCtrl.sSWStatus,
                  iCloseReqLoadGripperSh1 := "DB_LoaderShuttle1".sIntLoadUnload.oLoadGripperCloseReq OR "DB_LoaderShuttle1".sIntLoadUnloadOP.oLoadGripperCloseReq,
                  iCloseReqLoadGripperSh2 := "DB_LoaderShuttle2".sIntLoadUnload.oLoadGripperCloseReq OR "DB_LoaderShuttle2".sIntLoadUnloadOP.oLoadGripperCloseReq,
                  iCloseReqFixture := "DB_GestionFixture".sFixtureHold,
                  iDrilling_Finished := "DB_ScannerComm".oEndOfJob OR #sPosition.iDrilling_Finished,
                  iCloseReqUnloadGripper := "DB_GestionGripper".sUnloadGripperCloseReq,
                  iOpenReqUnloadGripperSh1 := "DB_LoaderShuttle1".sIntLoadUnload.oUnloadGripperOpenReq OR "DB_LoaderShuttle1".sIntLoadUnloadOP.oUnloadGripperOpenReq,
                  iOpenReqUnloadGripperSh2 := "DB_LoaderShuttle2".sIntLoadUnload.oUnloadGripperOpenReq OR "DB_LoaderShuttle2".sIntLoadUnloadOP.oUnloadGripperOpenReq,
                  iCondPartOutSh1 := (("DB_LoaderShuttle1".sExtLoadUnload.sInterface.JobDone AND NOT "DB_WorkingModes".sFilling) AND NOT "DB_WorkingModes".sSemiAuto) OR ( "DB_LoaderShuttle1".sExtLoadUnload.sCurrent_Step_NB = 150 AND "DB_WorkingModes".sSemiAuto),
                  iCondBwOutSh1 := "DB_LoaderShuttle1".sBwLoadUnload.sInterface.JobDone AND "DB_LoaderShuttle1".sBwLoadUnload.iUnloadReq,
                  iCondPartOutSh2 := (("DB_LoaderShuttle2".sExtLoadUnload.sInterface.JobDone AND NOT "DB_WorkingModes".sFilling) AND NOT "DB_WorkingModes".sSemiAuto) OR ( "DB_LoaderShuttle2".sExtLoadUnload.sCurrent_Step_NB = 150 AND "DB_WorkingModes".sSemiAuto),
                  iCondBwOutSh2 := "DB_LoaderShuttle2".sBwLoadUnload.sInterface.JobDone AND "DB_LoaderShuttle2".sBwLoadUnload.iUnloadReq);
   END_REGION
END_FUNCTION_BLOCK

FUNCTION_BLOCK "FB_StatusPart"   // FB87, SCL
{ S7_Optimized_Access := 'TRUE' }
// stored: MemoryReserve 100, SetENOAutomatically false
   VAR_INPUT
      iGood { ExternalAccessible := 'False'; ExternalVisible := 'False'; ExternalWritable := 'False'} : Bool;
      iUnknown { ExternalAccessible := 'False'; ExternalVisible := 'False'; ExternalWritable := 'False'} : Bool;
      iBad { ExternalAccessible := 'False'; ExternalVisible := 'False'; ExternalWritable := 'False'} : Bool;
      iAbsent { ExternalAccessible := 'False'; ExternalVisible := 'False'; ExternalWritable := 'False'} : Bool;
      iPresentUnexpected { ExternalAccessible := 'False'; ExternalVisible := 'False'; ExternalWritable := 'False'} : Bool;
      iAbsentUnexpected { ExternalAccessible := 'False'; ExternalVisible := 'False'; ExternalWritable := 'False'} : Bool;
   END_VAR
   VAR_OUTPUT
      oStatus { ExternalAccessible := 'False'; ExternalVisible := 'False'; ExternalWritable := 'False'} : "UDT_PartState";
   END_VAR
   VAR CONSTANT
      GOOD : Byte := 3;
      UNKNOW : Byte := 1;
      BAD : Byte := 2;
      ABSENT : Byte := 0;
      PRESENT_UNEXPECTED : Byte := 4;
      ABSENT_UNEXPECTED : Byte := 5;
      UNKNOW_STATUS : Byte := 99;
   END_VAR
BEGIN
   REGION Description header 
       //==================================================================================
       // POSALUX Swiss SA / (C) Copyright 2024
       //----------------------------------------------------------------------------------
       // Title: FB_StatusPart
       // Comment/Function: 
       //
       // Author: Fabien WALDT
       // Engineering: TIA Portal v20
       //----------------------------------------------------------------------------------
       // Change log table:
       // Version  | Date     | Expert in charge | Changes applied
       // ---------|----------|------------------|------------------------------------
       // 00.00.01 | 20251024 | WFA              | First released version
       // ==================================================================================
   END_REGION

   REGION Status
       #oStatus.Good := #iGood;
       #oStatus.Unknown := #iUnknown;
       #oStatus.Bad := #iBad;
       #oStatus.Absent := #iAbsent;
       #oStatus.PresentUnexpected := #iPresentUnexpected;
       #oStatus.AbsentUnexpected := #iAbsentUnexpected;
   END_REGION
END_FUNCTION_BLOCK

FUNCTION_BLOCK "FB_Position"   // FB38, SCL
{ S7_Optimized_Access := 'TRUE' }
// stored: MemoryReserve 100, SetENOAutomatically false
   VAR_INPUT
      iCondPartInSh1 : Bool;
      iCondBwInSh1 : Bool;
      iCondPartInSh2 : Bool;
      iCondBwInSh2 : Bool;
      iCondPartPresCtrlInSh1 : Bool;
      iCondBWPresCtrlInSh1 : Bool;
      iCondPartPresCtrlInSh2 : Bool;
      iCondBWPresCtrlInSh2 : Bool;
      iCondPartPresCtrlOutSh1 : Bool;
      iCondPartPresCtrlOutSh2 : Bool;
      iUndrilledPartPresence : Bool;
      iDrilledPartPresence : Bool;
      iUndrilledBWPresence : Bool;
      iCloseReqLoadGripperSh1 : Bool;
      iCloseReqLoadGripperSh2 : Bool;
      iCloseReqFixture : Bool;
      iDrilling_Finished : Bool;
      iCloseReqUnloadGripper : Bool;
      iOpenReqUnloadGripperSh1 : Bool;
      iOpenReqUnloadGripperSh2 : Bool;
      iCondPartOutSh1 : Bool;
      iCondBwOutSh1 : Bool;
      iCondPartOutSh2 : Bool;
      iCondBwOutSh2 : Bool;
   END_VAR
   VAR RETAIN
      sShuttle1 : "UDT_PartPosition";
      sShuttle2 { S7_SetPoint := 'True'} : "UDT_PartPosition";
      sGripper { S7_SetPoint := 'True'} : "UDT_PartPosition";
      sFixture { S7_SetPoint := 'True'} : "UDT_PartPosition";
   END_VAR
   VAR
      sRT_PartInSh1 : R_TRIG;
      sRT_BwInSh1 : R_TRIG;
      sRT_PartInSh2 : R_TRIG;
      sRT_BwInSh2 : R_TRIG;
      sRT_PartPresenceInSh1 { S7_SetPoint := 'True'} : R_TRIG;
      sRT_BWPresenceInSh1 { S7_SetPoint := 'True'} : R_TRIG;
      sRT_PartPresenceInSh2 { S7_SetPoint := 'True'} : R_TRIG;
      sRT_BWPresenceInSh2 { S7_SetPoint := 'True'} : R_TRIG;
      sRT_PartPresenceOutSh1 { S7_SetPoint := 'True'} : R_TRIG;
      sRT_PartPresenceOutSh2 { S7_SetPoint := 'True'} : R_TRIG;
      sRT_CloseLoadGripperSh1 : R_TRIG;
      sRT_CloseLoadGripperSh2 : R_TRIG;
      sRT_CloseFixture { S7_SetPoint := 'True'} : R_TRIG;
      sRT_Drilling_Finished { S7_SetPoint := 'True'} : R_TRIG;
      sRT_CloseUnloadGripper { S7_SetPoint := 'True'} : R_TRIG;
      sRT_OpenUnloadGripperSh1 { S7_SetPoint := 'True'} : R_TRIG;
      sRT_OpenUnloadGripperSh2 { S7_SetPoint := 'True'} : R_TRIG;
      sRT_PartOutSh1 : R_TRIG;
      sRT_BwOutSh1 : R_TRIG;
      sRT_PartOutSh2 : R_TRIG;
      sRT_BwOutSh2 : R_TRIG;
      sMachineEmpty { S7_SetPoint := 'True'} : Bool;
      sShuttle1Empty { S7_SetPoint := 'True'} : Bool;
      sShuttle2Empty { S7_SetPoint := 'True'} : Bool;
      sGripperEmpty { S7_SetPoint := 'True'} : Bool;
      sFixtureEmpty { S7_SetPoint := 'True'} : Bool;
      sPartNumber : Struct
         Shuttle1 : Int;
         Shuttle2 : Int;
         Gripper : Int;
         Fixture : Int;
         Total : Int;
      END_STRUCT;
      sEmptyPosition { S7_SetPoint := 'True'} : "UDT_EmptyPosition";
      sTON_PartPresenceOutSh1 { S7_SetPoint := 'True'} : TON_TIME;
      sTON_PartPresenceOutSh2 { S7_SetPoint := 'True'} : TON_TIME;
   END_VAR
BEGIN
   REGION Description header 
       //==================================================================================
       // POSALUX Swiss SA / (C) Copyright 2025
       //----------------------------------------------------------------------------------
       // Title: FB_Position
       // Comment/Function: 
       // Author: Fabien WALDT
       // Engineering: TIA Portal v17
       //----------------------------------------------------------------------------------
       // Change log table:
       // Version  | Date     | Expert in charge | Changes applied
       // ---------|----------|------------------|-----------------------------------------
       // 00.00.01 | 20250423 | WFA              | First released version
       // =================================================================================
   END_REGION

   REGION Input Part/BW Shuttle 1 (Loading)
       // Part
       #sRT_PartInSh1(CLK := #iCondPartInSh1);
       IF #sRT_PartInSh1.Q AND NOT "LBP_ModeGroup".E_JOG THEN
           #sShuttle1.Undrilled.Presence.Part := TRUE;
       END_IF;

       // BW
       #sRT_BwInSh1(CLK := #iCondBwInSh1);
       IF #sRT_BwInSh1.Q AND NOT "LBP_ModeGroup".E_JOG THEN
           #sShuttle1.Undrilled.Presence.BW := TRUE;
       END_IF;
   END_REGION

   REGION Input Part/BW Shuttle 2 (Loading)
       // Part
       #sRT_PartInSh2(CLK := #iCondPartInSh2);
       IF #sRT_PartInSh2.Q AND NOT "LBP_ModeGroup".E_JOG THEN
           #sShuttle2.Undrilled.Presence.Part := TRUE;
       END_IF;

       // BW
       #sRT_BwInSh2(CLK := #iCondBwInSh2);
       IF #sRT_BwInSh2.Q AND NOT "LBP_ModeGroup".E_JOG THEN
           #sShuttle2.Undrilled.Presence.BW := TRUE;
       END_IF;
   END_REGION

   REGION Input Part/BW Shuttle 1 (Control IN)
       // Part
       #sRT_PartPresenceInSh1(CLK := #iCondPartPresCtrlInSh1);
       IF #sRT_PartPresenceInSh1.Q AND NOT "LBP_ModeGroup".E_JOG THEN
           #sShuttle1.Undrilled.Presence.Part := #iUndrilledPartPresence;
           #sShuttle1.Drilled.Presence.Part := #iDrilledPartPresence;
       END_IF;

      // BW
       #sRT_BWPresenceInSh1(CLK := #iCondBWPresCtrlInSh1);
       IF #sRT_BWPresenceInSh1.Q AND NOT "LBP_ModeGroup".E_JOG THEN
           #sShuttle1.Undrilled.Presence.BW := #iUndrilledBWPresence;
       END_IF;
   END_REGION

   REGION Input Part/BW Shuttle 2 (Control IN)
       // Part
       #sRT_PartPresenceInSh2(CLK := #iCondPartPresCtrlInSh2);

       IF #sRT_PartPresenceInSh2.Q AND NOT "LBP_ModeGroup".E_JOG THEN
           #sShuttle2.Undrilled.Presence.Part := #iUndrilledPartPresence;
           #sShuttle2.Drilled.Presence.Part := #iDrilledPartPresence;
       END_IF;

       // BW
       #sRT_BWPresenceInSh2(CLK := #iCondBWPresCtrlInSh2);

       IF #sRT_BWPresenceInSh2.Q AND NOT "LBP_ModeGroup".E_JOG THEN
           #sShuttle2.Undrilled.Presence.BW := #iUndrilledBWPresence;
       END_IF;
   END_REGION

   REGION Transfert Shuttle 1/2 to Gripper U
       #sRT_CloseLoadGripperSh1(CLK := #iCloseReqLoadGripperSh1);
       #sRT_CloseLoadGripperSh2(CLK := #iCloseReqLoadGripperSh2);

       IF #sRT_CloseLoadGripperSh1.Q AND NOT "LBP_ModeGroup".E_JOG THEN
           #sGripper.Undrilled := #sShuttle1.Undrilled;
           #sShuttle1.Undrilled := #sEmptyPosition;
       ELSIF #sRT_CloseLoadGripperSh2.Q AND NOT "LBP_ModeGroup".E_JOG THEN
           #sGripper.Undrilled := #sShuttle2.Undrilled;
           #sShuttle2.Undrilled := #sEmptyPosition;
       END_IF;
   END_REGION

   REGION Transfert Gripper U to Fixture
       #sRT_CloseFixture(CLK := #iCloseReqFixture);

       IF #sRT_CloseFixture.Q AND NOT "LBP_ModeGroup".E_JOG THEN
           #sFixture.Undrilled :=  #sGripper.Undrilled;
           #sGripper.Undrilled := #sEmptyPosition;
       END_IF;
   END_REGION

   REGION Transfert Fixture Undrilled to Fixture Drilled
       #sRT_Drilling_Finished(CLK := #iDrilling_Finished);

       IF #sRT_Drilling_Finished.Q AND NOT "LBP_ModeGroup".E_JOG THEN
       #sFixture.Drilled := #sFixture.Undrilled;
           #sFixture.Undrilled := #sEmptyPosition;
       END_IF;
   END_REGION

   REGION Transfert Fixture to Gripper D
       #sRT_CloseUnloadGripper(CLK := #iCloseReqUnloadGripper);

       IF #sRT_CloseUnloadGripper.Q AND NOT "LBP_ModeGroup".E_JOG THEN
           #sGripper.Drilled := #sFixture.Drilled;
           #sFixture.Drilled := #sEmptyPosition;
       END_IF;
   END_REGION

   REGION Transfert Gripper D to Shuttle 1/2
       #sRT_OpenUnloadGripperSh1(CLK := #iOpenReqUnloadGripperSh1);
       #sRT_OpenUnloadGripperSh2(CLK := #iOpenReqUnloadGripperSh2);

       IF #sRT_OpenUnloadGripperSh1.Q AND NOT "LBP_ModeGroup".E_JOG THEN
           #sShuttle1.Drilled := #sGripper.Drilled;
           #sGripper.Drilled := #sEmptyPosition;
       ELSIF #sRT_OpenUnloadGripperSh2.Q AND NOT "LBP_ModeGroup".E_JOG THEN
           #sShuttle2.Drilled := #sGripper.Drilled;
           #sGripper.Drilled := #sEmptyPosition;
       END_IF;
   END_REGION

   REGION Output Part/BW Shuttle 1 (Unloading)
       // Part
       #sRT_PartOutSh1(CLK := #iCondPartOutSh1);
       IF #sRT_PartOutSh1.Q AND NOT "LBP_ModeGroup".E_JOG THEN
           #sShuttle1.Drilled.Presence.Part := FALSE;
       END_IF;

       // BW
       #sRT_BwOutSh1(CLK := #iCondBwOutSh1);
       IF #sRT_BwOutSh1.Q AND NOT "LBP_ModeGroup".E_JOG THEN
           #sShuttle1.Drilled.Presence.BW := FALSE;
       END_IF;
   END_REGION

   REGION Output Part/BW Shuttle 2 (Unloading)
       // Part
       #sRT_PartOutSh2(CLK := #iCondPartOutSh2);
       IF #sRT_PartOutSh2.Q AND NOT "LBP_ModeGroup".E_JOG THEN
           #sShuttle2.Drilled.Presence.Part := FALSE;
       END_IF;

       // BW
       #sRT_BwOutSh2(CLK := #iCondBwOutSh2);
       IF #sRT_BwOutSh2.Q AND NOT "LBP_ModeGroup".E_JOG THEN
           #sShuttle2.Drilled.Presence.BW := FALSE;
       END_IF;
   END_REGION

   REGION Output Part/BW Shuttle 1 (Control OUT)
       // Part
       #sTON_PartPresenceOutSh1(IN := #iCondPartPresCtrlOutSh1,
                                PT := t#100ms);

       #sRT_PartPresenceOutSh1(CLK := #sTON_PartPresenceOutSh1.Q);

       IF #sRT_PartPresenceOutSh1.Q AND NOT "LBP_ModeGroup".E_JOG THEN
           #sShuttle1.Undrilled.Presence.Part := #iUndrilledPartPresence;
           #sShuttle1.Drilled.Presence.Part := #iDrilledPartPresence;
       END_IF;

       // BW - No BW Control at output
   END_REGION

   REGION Output Part/BW Shuttle 2 (Control OUT)
       // Part
       #sTON_PartPresenceOutSh2(IN := #iCondPartPresCtrlOutSh2,
                                PT := t#100ms);

       #sRT_PartPresenceOutSh2(CLK := #iCondPartPresCtrlOutSh2);

       IF #sRT_PartPresenceOutSh2.Q AND NOT "LBP_ModeGroup".E_JOG THEN
           #sShuttle2.Undrilled.Presence.Part := #iUndrilledPartPresence;
           #sShuttle2.Drilled.Presence.Part := #iDrilledPartPresence;
       END_IF;

       // BW - No BW Control at output
   END_REGION

   REGION Machine states
       // Shuttle 1 Empty
       #sShuttle1Empty :=
       NOT #sShuttle1.Undrilled.Presence.Part
       AND NOT #sShuttle1.Undrilled.Presence.BW
       AND NOT #sShuttle1.Drilled.Presence.Part
       AND NOT #sShuttle1.Drilled.Presence.BW;

       // Shuttle 2 Empty
       #sShuttle2Empty :=
       NOT #sShuttle2.Undrilled.Presence.Part
       AND NOT #sShuttle2.Undrilled.Presence.BW
       AND NOT #sShuttle2.Drilled.Presence.Part
       AND NOT #sShuttle2.Drilled.Presence.BW;

       // Gripper Empty
       #sGripperEmpty :=
       NOT #sGripper.Undrilled.Presence.Part
       AND NOT #sGripper.Undrilled.Presence.BW
       AND NOT #sGripper.Drilled.Presence.Part
       AND NOT #sGripper.Drilled.Presence.BW;

       // Fixture Empty
       #sFixtureEmpty :=
       NOT #sFixture.Undrilled.Presence.Part
       AND NOT #sFixture.Undrilled.Presence.BW
       AND NOT #sFixture.Drilled.Presence.Part
       AND NOT #sFixture.Drilled.Presence.BW;

       // Machine Empty
       #sMachineEmpty := #sShuttle1Empty
       AND #sShuttle2Empty
       AND #sGripperEmpty
       AND #sFixtureEmpty;
   END_REGION

   REGION Part in Machine
       // Shuttle 1
       #sPartNumber.Shuttle1 := 0;
       IF #sShuttle1.Undrilled.Presence.Part AND #sShuttle1.Drilled.Presence.Part THEN
           #sPartNumber.Shuttle1 := 2;
       ELSIF #sShuttle1.Undrilled.Presence.Part XOR #sShuttle1.Drilled.Presence.Part THEN
           #sPartNumber.Shuttle1 := 1;
       END_IF;

       // Shuttle 2
       #sPartNumber.Shuttle2 := 0;
       IF #sShuttle2.Undrilled.Presence.Part AND #sShuttle2.Drilled.Presence.Part THEN
           #sPartNumber.Shuttle2 := 2;
       ELSIF #sShuttle2.Undrilled.Presence.Part XOR #sShuttle2.Drilled.Presence.Part THEN
           #sPartNumber.Shuttle2 := 1;
       END_IF;

       // Gripper
       #sPartNumber.Gripper := 0;
       IF #sGripper.Undrilled.Presence.Part AND #sGripper.Drilled.Presence.Part THEN
           #sPartNumber.Gripper := 2;
       ELSIF #sGripper.Undrilled.Presence.Part XOR #sGripper.Drilled.Presence.Part THEN
           #sPartNumber.Gripper := 1;
       END_IF;

       // Fixture
       #sPartNumber.Fixture := 0;
       IF #sFixture.Undrilled.Presence.Part OR #sFixture.Drilled.Presence.Part THEN
           #sPartNumber.Fixture := 1;
       END_IF;

       // Total
       #sPartNumber.Total := #sPartNumber.Shuttle1 + #sPartNumber.Shuttle2 + #sPartNumber.Gripper + #sPartNumber.Fixture;
   END_REGION
END_FUNCTION_BLOCK

FUNCTION_BLOCK "FB_BwLoader"   // FB88, SCL
{ S7_Optimized_Access := 'TRUE' }
// stored: MemoryReserve 100, SetENOAutomatically false
   VAR
      sBwCommunication : "FB_BwCommunication";
      sTONBW_CtrlInProgress { S7_SetPoint := 'True'} : TP_TIME;
   END_VAR
BEGIN
   REGION Description header 
       //==================================================================================
       // POSALUX Swiss SA / (C) Copyright 2024
       //----------------------------------------------------------------------------------
       // Title: FB_BwLoader
       // Comment/Function: 
       //
       // Author: Fabien WALDT
       // Engineering: TIA Portal v20
       //----------------------------------------------------------------------------------
       // Change log table:
       // Version  | Date     | Expert in charge | Changes applied
       // ---------|----------|------------------|------------------------------------
       // 00.00.01 | 20260127 | WFA              | First released version
       // ==================================================================================
   END_REGION

   REGION Inputs Update
       "DB_BwLoaderExchange".Inputs.LifeFlag := "AI_LifeFlag";
       IF NOT #sBwCommunication.oLifeFlagError THEN
           "DB_BwLoaderExchange".Inputs.JobDone := "DI_JobDone";
           "DB_BwLoaderExchange".Inputs.LockShuttle := "DI_LockShuttle";
           "DB_BwLoaderExchange".Inputs.DataSend := "AI_DataSend";
           "DB_BwLoaderExchange".Inputs.DataReceive := "AI_DataReceive";
           "DB_BwLoaderExchange".Inputs.NoEmergencyStopAtBwLoader := "DI_NoEmergencyStopAtBwLoader";
           "DB_BwLoaderExchange".Inputs.SafetyDoorsClosedAtBwLoader := "DI_SafetyDoorsClosedAtBwLoader";
           "DB_BwLoaderExchange".Inputs.BwInErrorState := "AI_BwInErrorState";
           "DB_BwLoaderExchange".Inputs.UndrilledPartControl := "DI_UndrilledPartControl";
           "DB_BwLoaderExchange".Inputs.DrilledPartControl := "DI_DrilledPartControl";
           "DB_BwLoaderExchange".Inputs.BackwallControl := "DI_BackwallControl";
           "DB_BwLoaderExchange".Inputs.BwLoaderInSafePos := "DI_BwLoaderInSafePos";
       ELSE
           "DB_BwLoaderExchange".Inputs.JobDone := FALSE;
           "DB_BwLoaderExchange".Inputs.LockShuttle := FALSE;
           "DB_BwLoaderExchange".Inputs.DataSend := 0;
           "DB_BwLoaderExchange".Inputs.DataReceive := 0;
           "DB_BwLoaderExchange".Inputs.NoEmergencyStopAtBwLoader := FALSE;
           "DB_BwLoaderExchange".Inputs.SafetyDoorsClosedAtBwLoader := FALSE;
           "DB_BwLoaderExchange".Inputs.BwInErrorState := 0;
           "DB_BwLoaderExchange".Inputs.UndrilledPartControl := FALSE;
           "DB_BwLoaderExchange".Inputs.DrilledPartControl := FALSE;
           "DB_BwLoaderExchange".Inputs.BackwallControl := FALSE;
           "DB_BwLoaderExchange".Inputs.BwLoaderInSafePos := FALSE;
       END_IF;
   END_REGION

   REGION
       #sBwCommunication(iShuttle1Load := "DB_LoaderShuttle1".sBwLoadUnload.oBwLoadReq,
                         iShuttle1Unload := "DB_LoaderShuttle1".sBwLoadUnload.oBwUnloadReq,
                         iShuttle2Load := "DB_LoaderShuttle2".sBwLoadUnload.oBwLoadReq,
                         iShuttle2Unload := "DB_LoaderShuttle2".sBwLoadUnload.oBwUnloadReq,
                         iFromBwLoaderLifeFlag := "DB_BwLoaderExchange".Inputs.LifeFlag,
                         iFromBwLoaderJobDone := "DB_BwLoaderExchange".Inputs.JobDone,
                         iFromBwLoaderLockShuttle := "DB_BwLoaderExchange".Inputs.LockShuttle,
                         iFromBwLoaderDatasR := "DB_BwLoaderExchange".Inputs.DataReceive,
                         iFromBwLoaderDatasS:="DB_BwLoaderExchange".Inputs.DataSend,
                         iBwInErrorState:="DB_BwLoaderExchange".Inputs.BwInErrorState,
                         oLoadJobDone => #sBwCommunication.oLoadJobDone,
                         oUnloadJobDone => #sBwCommunication.oUnloadJobDone,
                         oLifeFlagError => #sBwCommunication.oLifeFlagError,
                         ioToBwLoaderLifeFlag := "DB_BwLoaderExchange".Outputs.LifeFlag,
                         ioToBwLoaderLoaderRequest := "DB_BwLoaderExchange".Outputs.LoaderRequest,
                         ioToBwLoaderLockShuttle := "DB_BwLoaderExchange".Outputs.LockShuttle,
                         ioToBwLoaderDatas := "DB_BwLoaderExchange".Outputs.DataSend);
      END_REGION

      REGION Alarmes
          // Défaut communication Chargeur de Backwall
          IF #sBwCommunication.oLifeFlagError THEN
              "LBP_AlarmMsgs".UserA[03].A70UUxx[28] := TRUE;
          END_IF;

          // Défaut général Chargeur de Backwall
          "LBP_AlarmMsgs".UserA[03].A70UUxx[29] := #sBwCommunication.iBwInErrorState <> 0;
      END_REGION

      REGION Outputs management
          "DB_BwLoaderExchange".Outputs.NoEmergencyStopAtFemto := NOT "DB_DataFromSafety".EmergencyStop;
          "DB_BwLoaderExchange".Outputs.SafetyDoorsClosedAtFemto := "DB_DataFromSafety".DoorsClosed;

          IF "DB_Alarms".sAlarmsLevel6 THEN
              "DB_BwLoaderExchange".Outputs.FemtoInErrorState := 6;
          ELSIF "DB_Alarms".sAlarmsLevel5 THEN
              "DB_BwLoaderExchange".Outputs.FemtoInErrorState := 5;
          ELSIF "DB_Alarms".sAlarmsLevel4 THEN
              "DB_BwLoaderExchange".Outputs.FemtoInErrorState := 4;
          ELSIF "DB_Alarms".sAlarmsLevel3 THEN
              "DB_BwLoaderExchange".Outputs.FemtoInErrorState := 3;
          ELSIF "DB_Alarms".sAlarmsLevel2 THEN
              "DB_BwLoaderExchange".Outputs.FemtoInErrorState := 2;
          ELSIF "DB_Alarms".sAlarmsLevel1 THEN
              "DB_BwLoaderExchange".Outputs.FemtoInErrorState := 1;
          ELSE
              "DB_BwLoaderExchange".Outputs.FemtoInErrorState := 1;
          END_IF;

          "DB_BwLoaderExchange".Outputs.AutoMode := "LBP_ModeGroup".E_AUTO;
          "DB_BwLoaderExchange".Outputs.JogMode := "LBP_ModeGroup".E_JOG;
          "DB_BwLoaderExchange".Outputs.GotoSafePos := "LBP_Chan1".A_Ref;
          "DB_BwLoaderExchange".Outputs.Emptying := "DB_WorkingModes".sEmptying;
      END_REGION

      REGION BW Control IN in progress
          "DB_BwLoaderExchange".Outputs.BW_CtrlInProgress :=
          ("DB_AxisPosition".sAxis05_U1."$AA_IM" = "DB_AxisPosMachinePLC".Axis_U1.BwControl AND "DB_LoaderShuttle1".sBwControlIn.sCurrent_Step_NB <> 0)
          OR ("DB_AxisPosition".sAxis06_U2."$AA_IM" = "DB_AxisPosMachinePLC".Axis_U2.BwControl AND "DB_LoaderShuttle2".sBwControlIn.sCurrent_Step_NB <> 0);
      END_REGION

      REGION  Outputs Update
          "AQ_LifeFlag" := "DB_BwLoaderExchange".Outputs.LifeFlag;
          "DQ_LoaderRequest":= "DB_BwLoaderExchange".Outputs.LoaderRequest;
          "DQ_LockShuttle" := "DB_BwLoaderExchange".Outputs.LockShuttle;
          "AQ_DataSend" := "DB_BwLoaderExchange".Outputs.DataSend;
          "AQ_DataReceive":= "DB_BwLoaderExchange".Outputs.DataReceive;
          "DQ_NoEmergencyStopAtFemto" := "DB_BwLoaderExchange".Outputs.NoEmergencyStopAtFemto;
          "DQ_SafetyDoorsClosedAtFemto" := "DB_BwLoaderExchange".Outputs.SafetyDoorsClosedAtFemto;
          "AQ_FemtoInErrorState" := "DB_BwLoaderExchange".Outputs.FemtoInErrorState;
          "DQ_AutoMode" :="DB_BwLoaderExchange".Outputs.AutoMode;
          "DQ_JogMode" := "DB_BwLoaderExchange".Outputs.JogMode;
          "DQ_GotoSafePos":= "DB_BwLoaderExchange".Outputs.GotoSafePos;
          "DQ_Emptying" := "DB_BwLoaderExchange".Outputs.Emptying;
          "DQ_BW_CtrlInProgress" := "DB_BwLoaderExchange".Outputs.BW_CtrlInProgress;
      END_REGION

      REGION Reset à supprimer
          IF "DB_McpKeyboardSignals".sAlarmReset.sKeySWStatus THEN
              "AQ_Reset" := 1;
          ELSIF "MCP1_In".reset THEN
              "AQ_Reset" := 2;
          ELSE
              "AQ_Reset" := 0;
          END_IF;
      END_REGION
END_FUNCTION_BLOCK

FUNCTION_BLOCK "FB_BwCommunication"   // FB71, SCL
{ S7_Optimized_Access := 'TRUE' }
// stored: MemoryReserve 100, SetENOAutomatically false
   VAR_INPUT
      iShuttle1Load : Bool;
      iShuttle1Unload : Bool;
      iShuttle2Load : Bool;
      iShuttle2Unload : Bool;
      iFromBwLoaderLifeFlag : Int;
      iFromBwLoaderJobDone : Bool;
      iFromBwLoaderLockShuttle : Bool;
      iFromBwLoaderDatasR : Int;
      iFromBwLoaderDatasS : Int;
      iBwInErrorState : Int;
   END_VAR
   VAR_OUTPUT
      oLifeFlagError : Bool;
      oLoadJobDone : Bool;
      oUnloadJobDone : Bool;
   END_VAR
   VAR_IN_OUT
      ioToBwLoaderLifeFlag : Int;
      ioToBwLoaderLoaderRequest { ExternalAccessible := 'False'; ExternalVisible := 'False'; ExternalWritable := 'False'} : Bool;
      ioToBwLoaderLockShuttle { ExternalAccessible := 'False'; ExternalVisible := 'False'; ExternalWritable := 'False'} : Bool;
      ioToBwLoaderDatas { ExternalAccessible := 'False'; ExternalVisible := 'False'; ExternalWritable := 'False'} : Int;
   END_VAR
   VAR
      sPrevLifeFlagFrom : Int;
      sTimerWatchdogCtrl : TON_TIME;
      sRT_1Hz { S7_SetPoint := 'True'} : R_TRIG;
      sShuttle1Locked { S7_SetPoint := 'True'} : Bool;
      sShuttle2Locked : Bool;
      sStep : Int;
      sRT_Shuttle1Load : R_TRIG;
      sRT_Shuttle1Unload : R_TRIG;
      sRT_Shuttle2Load : R_TRIG;
      sRT_Shuttle2Unload : R_TRIG;
   END_VAR
   VAR CONSTANT
      ID_SHUTTLE1_LOAD : Int := 101;
      ID_SHUTTLE1_UNLOAD : Int := 102;
      ID_SHUTTLE2_LOAD : Int := 201;
      ID_SHUTTLE2_UNLOAD : Int := 202;
   END_VAR
BEGIN
   REGION Description header 
       //==================================================================================
       // POSALUX Swiss SA / (C) Copyright 2024
       //----------------------------------------------------------------------------------
       // Title: 
       // Comment/Function: 
       //
       // Author: Fabien WALDT
       // Engineering: TIA Portal v20
       //----------------------------------------------------------------------------------
       // Change log table:
       // Version  | Date     | Expert in charge | Changes applied
       // ---------|----------|------------------|------------------------------------
       // 00.00.01 | 20260127 | WFA              | First released version
       // ==================================================================================
   END_REGION

   REGION Increment LifeFlag
       #sRT_1Hz(CLK := "Clock_1Hz");

       IF #sRT_1Hz.Q THEN
           #ioToBwLoaderLifeFlag := #ioToBwLoaderLifeFlag + 1;
       END_IF;

       IF #ioToBwLoaderLifeFlag < 0 OR #ioToBwLoaderLifeFlag > 59 THEN
           #ioToBwLoaderLifeFlag := 0;
       END_IF;
   END_REGION

   REGION Commm Control
       // Lancement du timer de controle
       #sTimerWatchdogCtrl(IN := #iFromBwLoaderLifeFlag = #sPrevLifeFlagFrom,
                           PT := T#2s);

       // Check value change
       #oLifeFlagError := FALSE;
       IF #sTimerWatchdogCtrl.Q THEN
           #oLifeFlagError := TRUE;
       END_IF;
       // Save current value
       #sPrevLifeFlagFrom := #iFromBwLoaderLifeFlag;
   END_REGION

   REGION Init
       IF  NOT #iShuttle1Load AND NOT #iShuttle1Unload AND NOT #iShuttle2Load AND NOT #iShuttle2Unload THEN
           #ioToBwLoaderDatas := 0;
               #ioToBwLoaderLoaderRequest := FALSE;
           END_IF;
   END_REGION

   REGION R_Trig Load/Unload
       #sRT_Shuttle1Load(CLK := #iShuttle1Load);
       #sRT_Shuttle1Unload(CLK := #iShuttle1Unload);
       #sRT_Shuttle2Load(CLK := #iShuttle2Load);
       #sRT_Shuttle2Unload(CLK := #iShuttle2Unload);
   END_REGION

   REGION Commm sequence

       IF NOT #oLifeFlagError THEN
           // Send Job Request
           IF #iBwInErrorState = 0 THEN
               IF #sRT_Shuttle1Load.Q THEN
                   #ioToBwLoaderDatas := #ID_SHUTTLE1_LOAD;
                   #ioToBwLoaderLoaderRequest := TRUE;
               ELSIF #sRT_Shuttle1Unload.Q THEN
                   #ioToBwLoaderDatas := #ID_SHUTTLE1_UNLOAD;
                   #ioToBwLoaderLoaderRequest := TRUE;
               ELSIF #sRT_Shuttle2Load.Q THEN
                   #ioToBwLoaderDatas := #ID_SHUTTLE2_LOAD;
                   #ioToBwLoaderLoaderRequest := TRUE;
               ELSIF #sRT_Shuttle2Unload.Q THEN
                   #ioToBwLoaderDatas := #ID_SHUTTLE2_UNLOAD;
                   #ioToBwLoaderLoaderRequest := TRUE;
               END_IF;
           END_IF;
           // Send Shuttle locked to BW
           IF #ioToBwLoaderDatas = #ID_SHUTTLE1_LOAD OR #ioToBwLoaderDatas = #ID_SHUTTLE1_UNLOAD THEN
               #ioToBwLoaderLockShuttle := "LBP_Axis05_U1".A_FDSpStop AND #iFromBwLoaderLockShuttle;
           ELSIF #ioToBwLoaderDatas = #ID_SHUTTLE2_LOAD OR #ioToBwLoaderDatas = #ID_SHUTTLE2_UNLOAD THEN
               #ioToBwLoaderLockShuttle := "LBP_Axis06_U2".A_FDSpStop AND #iFromBwLoaderLockShuttle;
               "DB_WAF".bSpy[12] := TRUE;
           ELSE
               #ioToBwLoaderLockShuttle := FALSE;
           END_IF;

           // Send Locked shuttle to axis
           IF #ioToBwLoaderLoaderRequest AND #iFromBwLoaderLockShuttle THEN
               #sShuttle1Locked := TRUE;
               #sShuttle2Locked := TRUE;
           ELSE
               #sShuttle1Locked := FALSE;
               #sShuttle2Locked := FALSE;
           END_IF;

          // Job Done
           IF #iFromBwLoaderJobDone AND (#iFromBwLoaderDatasS = #ID_SHUTTLE1_LOAD OR #iFromBwLoaderDatasS = #ID_SHUTTLE2_LOAD) THEN
               #oLoadJobDone := TRUE;
               IF "DB_LoaderShuttle1".sBwLoadUnload.sCurrent_Step_NB <> 50 AND "DB_LoaderShuttle2".sBwLoadUnload.sCurrent_Step_NB <> 50 THEN
                   #ioToBwLoaderLoaderRequest := FALSE;
               END_IF;
           ELSIF #iFromBwLoaderJobDone AND (#iFromBwLoaderDatasS = #ID_SHUTTLE1_UNLOAD OR #iFromBwLoaderDatasS = #ID_SHUTTLE2_UNLOAD) THEN
               #oUnloadJobDone := TRUE;
               IF "DB_LoaderShuttle1".sBwLoadUnload.sCurrent_Step_NB <> 150 AND "DB_LoaderShuttle2".sBwLoadUnload.sCurrent_Step_NB <> 150 THEN
                   #ioToBwLoaderLoaderRequest := FALSE;
               END_IF;
           ELSE
               #oLoadJobDone := FALSE;
               #oUnloadJobDone := FALSE;
           END_IF;
       END_IF;
   END_REGION
END_FUNCTION_BLOCK

FUNCTION_BLOCK "FB_GestionWorkingModes"   // FB94, SCL
{ S7_Optimized_Access := 'TRUE' }
// stored: MemoryReserve 100, SetENOAutomatically false
   VAR
      sMCP_KxxKeysDisable : Bool;
   END_VAR
BEGIN
   REGION Description header 
       //==================================================================================
       // POSALUX Swiss SA / (C) Copyright 2025
       //----------------------------------------------------------------------------------
       // Title: FB_GestionWorkingModes
       // Comment/Function: 
       // Author: Fabien WALDT
       // Engineering: TIA Portal v17
       //----------------------------------------------------------------------------------
       // Change log table:
       // Version  | Date     | Expert in charge | Changes applied
       // ---------|----------|------------------|-----------------------------------------
       // 00.00.01 | 20251218 | WFA              | First released version
       // =================================================================================
   END_REGION

   REGION Working Modes
       // MCP Keys Auto - Semi Auto disable
       "DB_McpKeyboardSignals".sK10_LoaderAuto.sKeyDisable := NOT "DB_WorkingModes".iChangeModeEnable OR #sMCP_KxxKeysDisable;
       "DB_McpKeyboardSignals".sK11_LoaderSemiAuto.sKeyDisable := NOT "DB_WorkingModes".iChangeModeEnable OR #sMCP_KxxKeysDisable;

       // Auto Mode Request
       IF "DB_McpKeyboardSignals".sK10_LoaderAuto.sKeySWTogglePositiveFront
           OR "DB_OPC_State".sRT_AutoReq.Q THEN
           "DB_WorkingModes".ioAutoReq := TRUE;
           "DB_McpKeyboardSignals".sK10_LoaderAuto.sKeySWToggleStatus := TRUE;
           "DB_McpKeyboardSignals".sK11_LoaderSemiAuto.sKeySWToggleStatus := FALSE;
       END_IF;

       // Semi Auto Mode Request
       IF "DB_McpKeyboardSignals".sK11_LoaderSemiAuto.sKeySWTogglePositiveFront
           OR "DB_OPC_State".sRT_SemiAutoReq.Q THEN
           "DB_WorkingModes".ioSemiAutoReq := TRUE;
           "DB_McpKeyboardSignals".sK10_LoaderAuto.sKeySWToggleStatus := FALSE;
           "DB_McpKeyboardSignals".sK11_LoaderSemiAuto.sKeySWToggleStatus := TRUE;
       END_IF;

       // Manu Mode Request
       IF ("DB_McpKeyboardSignals".sK11_LoaderSemiAuto.sKeySWToggleNegativeFront AND NOT "DB_McpKeyboardSignals".sK10_LoaderAuto.sKeySWToggleStatus)
           OR ("DB_McpKeyboardSignals".sK10_LoaderAuto.sKeySWToggleNegativeFront AND NOT "DB_McpKeyboardSignals".sK11_LoaderSemiAuto.sKeySWToggleStatus)
           OR "DB_OPC_State".sRT_ManuReq.Q THEN
           "DB_WorkingModes".ioManuReq := TRUE;
           "DB_McpKeyboardSignals".sK10_LoaderAuto.sKeySWToggleStatus := FALSE;
           "DB_McpKeyboardSignals".sK11_LoaderSemiAuto.sKeySWToggleStatus := FALSE;
       END_IF;

       "DB_WorkingModes"(ioEmptyingReq := "DB_HMISetting".WorkingMode.EmptyingReq,
                         ioAutoReq := "DB_WorkingModes".ioAutoReq,
                         ioSemiAutoReq := "DB_WorkingModes".ioSemiAutoReq,
                         ioManuReq := "DB_WorkingModes".ioManuReq,
                         iChangeModeEnable := NOT "DB_LoaderShuttle1".sMain.sInterface.SequenceRun
                         AND NOT "DB_LoaderShuttle2".sMain.sInterface.SequenceRun);

       IF "DB_PartManagement".sPosition.sMachineEmpty THEN
           "DB_HMISetting".WorkingMode.EmptyingReq := FALSE;
       END_IF;

       // Reset flags OPC
       "DB_OPC_State".sAutoReq := FALSE;
       "DB_OPC_State".sSemiAutoReq := FALSE;
       "DB_OPC_State".sManuReq := FALSE;
   END_REGION

   REGION Kxx Keys Disable
       IF #sMCP_KxxKeysDisable THEN
           "DB_McpKeyboardSignals".sK1_Powermeter.sKeyDisable := TRUE;
           "DB_McpKeyboardSignals".sK2_GasAssist.sKeyDisable := TRUE;
           "DB_McpKeyboardSignals".sK3_KeySaveParam.sKeyDisable := TRUE;
           "DB_McpKeyboardSignals".sK4_GripperUndrilledPart.sKeyDisable := TRUE;
           "DB_McpKeyboardSignals".sK5_GripperDrilledPart.sKeyDisable := TRUE;
           "DB_McpKeyboardSignals".sK6_SITestStop.sKeyDisable := TRUE;
           "DB_McpKeyboardSignals".sK7_FixtureClamp.sKeyDisable := TRUE;
           "DB_McpKeyboardSignals".sK8_FixtureVacuum.sKeyDisable := TRUE;
           "DB_McpKeyboardSignals".sK9_Aspiration.sKeyDisable := TRUE;
           "DB_McpKeyboardSignals".sK10_LoaderAuto.sKeyDisable := TRUE;
           "DB_McpKeyboardSignals".sK11_LoaderSemiAuto.sKeyDisable := TRUE;
           "DB_McpKeyboardSignals".sK12_ObservationCamera.sKeyDisable := TRUE;
           "DB_McpKeyboardSignals".sK13_MainDoor.sKeyDisable := TRUE;
           "DB_McpKeyboardSignals".sK14_WarmUp.sKeyDisable := TRUE;
           "DB_McpKeyboardSignals".sK15_MachineLight.sKeyDisable := TRUE;
       END_IF;
   END_REGION
END_FUNCTION_BLOCK

FUNCTION_BLOCK "FB_WorkingModes"   // FB56, SCL
{ S7_Optimized_Access := 'TRUE' }
// stored: MemoryReserve 100, SetENOAutomatically false
   VAR_INPUT
      iChangeModeEnable : Bool;
   END_VAR
   VAR_IN_OUT
      ioEmptyingReq : Bool;
      ioAutoReq : Bool;
      ioSemiAutoReq : Bool;
      ioManuReq : Bool;
   END_VAR
   VAR
      sRT_Filling : R_TRIG;
      sRT_Normal { S7_SetPoint := 'True'} : R_TRIG;
      sRT_Emptying { S7_SetPoint := 'True'} : R_TRIG;
      sFT_Emptying { S7_SetPoint := 'True'} : F_TRIG;
      sRT_Auto { S7_SetPoint := 'True'} : R_TRIG;
      sRT_SemiAuto { S7_SetPoint := 'True'} : R_TRIG;
      sRT_Manu { S7_SetPoint := 'True'} : R_TRIG;
      sFilling { S7_SetPoint := 'True'} : Bool;
      sNormal : Bool;
      sEmptying : Bool;
      sAuto : Bool;
      sSemiAuto : Bool;
      sManu : Bool;
      sOnePiece : Bool;
      sDryRun : Bool;
   END_VAR
BEGIN
   REGION Description header 
       //==================================================================================
       // POSALUX Swiss SA / (C) Copyright 2025
       //----------------------------------------------------------------------------------
       // Title: FB_WorkingModes
       // Comment/Function: 
       // Author: Fabien WALDT
       // Engineering: TIA Portal v17
       //----------------------------------------------------------------------------------
       // Change log table:
       // Version  | Date     | Expert in charge | Changes applied
       // ---------|----------|------------------|-----------------------------------------
       // 00.00.01 | 20251218 | WFA              | First released version
       // =================================================================================
   END_REGION

   REGION Filling - Normal - Emptying
       #sRT_Emptying(CLK := #ioEmptyingReq);
       #sFT_Emptying(CLK := #ioEmptyingReq);

       #sRT_Filling(CLK := ("DB_LoaderShuttle1".sMain.iJobReq OR "DB_LoaderShuttle2".sMain.iJobReq)
                    AND "DB_PartManagement".sPosition.sMachineEmpty AND NOT #sEmptying);

       #sRT_Normal(CLK := (("DB_LoaderShuttle1".sMain.iJobReq OR "DB_LoaderShuttle2".sMain.iJobReq)
                   AND NOT "DB_PartManagement".sPosition.sMachineEmpty
                   AND NOT #sFilling)
                   OR ("DB_PartManagement".sPosition.sFixture.Drilled.Presence.Part AND NOT #sNormal AND NOT #sEmptying)
                   OR #sFT_Emptying.Q);

       IF #sRT_Filling.Q THEN
           #sFilling := TRUE;
           #sNormal := FALSE;
           #sEmptying := FALSE;
       END_IF;

       IF #sRT_Normal.Q THEN
           #sFilling := FALSE;
           #sNormal := TRUE;
           #sEmptying := FALSE;
       END_IF;

       IF #sRT_Emptying.Q THEN
           #sFilling := FALSE;
           #sNormal := FALSE;
           #sEmptying := TRUE;
       END_IF;
   END_REGION

   REGION Auto - Semi Auto - Manu
       #sRT_Auto(CLK := #ioAutoReq OR (NOT #sAuto AND NOT #sSemiAuto AND NOT #sManu));
       #sRT_SemiAuto(CLK := #ioSemiAutoReq);
       #sRT_Manu(CLK := #ioManuReq);

       IF #iChangeModeEnable THEN
           IF #sRT_Auto.Q THEN
               #sAuto := TRUE;
               #sSemiAuto := FALSE;
               #sManu := FALSE;
           ELSIF #sRT_SemiAuto.Q THEN
               #sAuto := FALSE;
               #sSemiAuto := TRUE;
               #sManu := FALSE;
           ELSIF #sRT_Manu.Q THEN
               #sAuto := FALSE;
               #sSemiAuto := FALSE;
               #sManu := TRUE;
           END_IF;
       END_IF;

       #ioAutoReq := FALSE;
       #ioSemiAutoReq := FALSE;
       #ioManuReq := FALSE;
   END_REGION
END_FUNCTION_BLOCK

FUNCTION_BLOCK "FB_Simulation"   // FB48, SCL
{ S7_Optimized_Access := 'TRUE' }
// stored: MemoryReserve 100, SetENOAutomatically false
   VAR
      sExtLoadUnloadTimer1 : TON_TIME;
      sExtLoadUnloadTimer2 { S7_SetPoint := 'True'} : TON_TIME;
      sBwLoadUnloadTimer1 { S7_SetPoint := 'True'} : TON_TIME;
      sBwLoadUnloadTimer2 { S7_SetPoint := 'True'} : TON_TIME;
      sTON_UndrilledGripperFull { S7_SetPoint := 'True'} : TON_TIME;
      sTON_UndrilledFixture { S7_SetPoint := 'True'} : TON_TIME;
      sTON_DrilledFixture { S7_SetPoint := 'True'} : TON_TIME;
      sTON_ResetBit { S7_SetPoint := 'True'} : TON_TIME;
      sSeqRun { S7_SetPoint := 'True'} : Bool;
      sTON_CloseDrilledGripper_1 { S7_SetPoint := 'True'} : TON_TIME;
      sTONCloseFixture { S7_SetPoint := 'True'} : TON_TIME;
      sTONOpenFixture { S7_SetPoint := 'True'} : TON_TIME;
      sTONOpenFixture1 { S7_SetPoint := 'True'} : TON_TIME;
      sTON_CloseDrilledGripper { S7_SetPoint := 'True'} : TON_TIME;
      sTON_WorkinProgress { S7_SetPoint := 'True'} : TON_TIME;
      sTON_OpenUndrilledGripper { S7_SetPoint := 'True'} : TON_TIME;
      sRT_NC_Mode { S7_SetPoint := 'True'} : R_TRIG;
      sStep { S7_SetPoint := 'True'} : Array[0..15] of Bool;
      sRT_DrillingFinished : R_TRIG;
      "sTON_No MCodes" { S7_SetPoint := 'True'} : TON_TIME;
      sRT_TONMCodes { S7_SetPoint := 'True'} : R_TRIG;
      sRT_FIXLoading { S7_SetPoint := 'True'} : R_TRIG;
      sRT_FIXblowing { S7_SetPoint := 'True'} : R_TRIG;
      sRT_MemoLoaderStart { S7_SetPoint := 'True'} : R_TRIG;
      sRT_Sh1_ExtLoadUnloadDone { S7_SetPoint := 'True'} : R_TRIG;
      sRT_Sh2_ExtLoadUnloadDone { S7_SetPoint := 'True'} : R_TRIG;
   END_VAR
BEGIN
   REGION Ext Load/Unload Time
       // Necessaire pour Dry Run
       #sExtLoadUnloadTimer1(IN:= "DB_LoaderShuttle1".sExtLoadUnload.sCurrent_Step_NB = 50
                             OR "DB_LoaderShuttle1".sExtLoadUnload.sCurrent_Step_NB = 80
                             OR "DB_LoaderShuttle1".sExtLoadUnload.sCurrent_Step_NB = 110,
                             PT:= t#3s);
      "DB_SonplasMain".sSonplasLoader.iPartInShuttle1Finished := #sExtLoadUnloadTimer1.Q;

      #sExtLoadUnloadTimer2(IN :=  "DB_LoaderShuttle2".sExtLoadUnload.sCurrent_Step_NB = 50
                            OR "DB_LoaderShuttle2".sExtLoadUnload.sCurrent_Step_NB = 80
                            OR "DB_LoaderShuttle2".sExtLoadUnload.sCurrent_Step_NB = 110,
                            PT := t#3s);
      "DB_SonplasMain".sSonplasLoader.iPartInShuttle2Finished := #sExtLoadUnloadTimer2.Q;
   END_REGION

   REGION Bw Load/Unload Time
       // Necessaire pour Dry Run
       #sBwLoadUnloadTimer1(IN := "DB_LoaderShuttle1".sBwLoadUnload.sCurrent_Step_NB = 50
                            OR "DB_LoaderShuttle1".sBwLoadUnload.sCurrent_Step_NB = 150,
                            PT := t#2s);

       #sBwLoadUnloadTimer2(IN := "DB_LoaderShuttle2".sBwLoadUnload.sCurrent_Step_NB = 50
                            OR "DB_LoaderShuttle2".sBwLoadUnload.sCurrent_Step_NB = 150,
                            PT := t#2s);
       "DB_BwLoader".sBwCommunication.oLoadJobDone := #sBwLoadUnloadTimer1.Q OR #sBwLoadUnloadTimer2.Q;
      "DB_BwLoader".sBwCommunication.oUnloadJobDone := #sBwLoadUnloadTimer1.Q OR #sBwLoadUnloadTimer2.Q;
   END_REGION

   REGION Part Position  
      // Necessaire pour Dry Run
       IF ("DB_LoaderShuttle1".sControlIn.sInterface.SequenceRun OR "DB_LoaderShuttle2".sControlIn.sInterface.SequenceRun) AND NOT "DB_WAF".CtrlInEnable THEN
          IF "DB_WorkingModes".sFilling THEN
              "DB_DigitalInputsBW_Station".sUndrilledPartCtrl.sSWStatus := TRUE;
              "DB_DigitalInputsBW_Station".sDrilledPartCtrl.sSWStatus := FALSE;
          ELSIF "DB_WorkingModes".sNormal THEN
              "DB_DigitalInputsBW_Station".sUndrilledPartCtrl.sSWStatus := TRUE;
              "DB_DigitalInputsBW_Station".sDrilledPartCtrl.sSWStatus := FALSE;
          ELSIF "DB_WorkingModes".sEmptying THEN
              "DB_DigitalInputsBW_Station".sUndrilledPartCtrl.sSWStatus := FALSE;
              "DB_DigitalInputsBW_Station".sDrilledPartCtrl.sSWStatus := FALSE;
          END_IF;
      END_IF;

      IF ("DB_LoaderShuttle1".sControlOut.sInterface.SequenceRun OR "DB_LoaderShuttle2".sControlOut.sInterface.SequenceRun) AND NOT "DB_WAF".CtrlOutEnable THEN
          IF "DB_WorkingModes".sFilling THEN
              "DB_DigitalInputsBW_Station".sUndrilledPartCtrl.sSWStatus := FALSE;
              "DB_DigitalInputsBW_Station".sDrilledPartCtrl.sSWStatus := FALSE;
          ELSIF "DB_WorkingModes".sNormal THEN
              "DB_DigitalInputsBW_Station".sUndrilledPartCtrl.sSWStatus := FALSE;
              "DB_DigitalInputsBW_Station".sDrilledPartCtrl.sSWStatus := TRUE;
          ELSIF "DB_WorkingModes".sEmptying THEN
              "DB_DigitalInputsBW_Station".sUndrilledPartCtrl.sSWStatus := FALSE;
              "DB_DigitalInputsBW_Station".sDrilledPartCtrl.sSWStatus := TRUE;
          END_IF;
      END_IF;
    END_REGION

    REGION BW Position
        // Necessaire pour Dry Run
        IF NOT "DB_WAF".CtrlBwEnable THEN
            IF "DB_WorkingModes".sNormal THEN
                "DB_DigitalInputsBW_Station".sBwCtrl.sSWStatus := TRUE;
            ELSIF "DB_WorkingModes".sEmptying THEN
                // "DB_DigitalInputsBW_Station".sBwCtrl.sSWStatus := FALSE;
                "DB_DigitalInputsBW_Station".sBwCtrl.sSWStatus := "DB_PartManagement".sPosition.sShuttle1.Undrilled.Presence.Part
                OR "DB_PartManagement".sPosition.sShuttle1.Undrilled.Presence.Part;
            ELSIF "DB_WorkingModes".sFilling THEN
                "DB_DigitalInputsBW_Station".sBwCtrl.sSWStatus := TRUE;
            END_IF;
        END_IF;
        END_REGION

   REGION Drilling Finished
      // Necessaire pour Dry Run
       #sRT_DrillingFinished(CLK := "DB_PartManagement".sPosition.sFixture.Undrilled.Presence.Part AND "DB_PartManagement".sPosition.sFixture.Undrilled.Presence.BW);
       "DB_PartManagement".sPosition.iDrilling_Finished := #sRT_DrillingFinished.Q;
   END_REGION

   REGION Interlock
      "DB_WAF".Sonplas.OperateInOutCollision := TRUE;
      "DB_WAF".BwLoader.Safe := TRUE;
      "DB_WAF".bSpy[9] := "DB_WAF".bSpy[9];
   END_REGION

   REGION Ext Loader
       "DB_LoaderOptions".ExtLoadUnload.Disabled := TRUE;

       #sRT_Sh1_ExtLoadUnloadDone(CLK := "DB_LoaderShuttle1".sExtLoadUnload.sInterface.JobDone);
       #sRT_Sh2_ExtLoadUnloadDone(CLK := "DB_LoaderShuttle2".sExtLoadUnload.sInterface.JobDone);

       IF #sRT_Sh1_ExtLoadUnloadDone.Q THEN
           "DB_SonplasMain".sSonplasLoader.iPartInDMC_CodeShuttle1[0] := "DB_SonplasMain".sSonplasLoader.iPartInDMC_CodeShuttle1[0] + 1;
           IF "DB_SonplasMain".sSonplasLoader.iPartInDMC_CodeShuttle1[0] > 99 THEN
               "DB_SonplasMain".sSonplasLoader.iPartInDMC_CodeShuttle1[0] := 0;
           END_IF;
       END_IF;

       IF #sRT_Sh2_ExtLoadUnloadDone.Q THEN
           "DB_SonplasMain".sSonplasLoader.iPartInDMC_CodeShuttle2[0] := "DB_SonplasMain".sSonplasLoader.iPartInDMC_CodeShuttle2[0] + 1;
           IF "DB_SonplasMain".sSonplasLoader.iPartInDMC_CodeShuttle2[0] > 99 THEN
               "DB_SonplasMain".sSonplasLoader.iPartInDMC_CodeShuttle2[0] := 0;
           END_IF;
       END_IF;
   END_REGION

   // REGION Shuttle Enable
   //     "DB_HMISetting".Shuttle1Enable := TRUE;
   //     "DB_HMISetting".Shuttle2Enable := TRUE;
   // END_REGION

   REGION Misc
          "DB_WorkingModes".sDryRun := FALSE;
   END_REGION

   REGION Reset Part Position
       IF "DB_WAF".ResetPartPosition THEN
           "DB_PartManagement".sPosition.sShuttle1.Undrilled.Presence.Part := FALSE;
           "DB_PartManagement".sPosition.sShuttle1.Undrilled.Presence.BW := FALSE;
           "DB_PartManagement".sPosition.sShuttle1.Drilled.Presence.Part := FALSE;
           "DB_PartManagement".sPosition.sShuttle1.Drilled.Presence.BW := FALSE;

           "DB_PartManagement".sPosition.sShuttle2.Undrilled.Presence.Part := FALSE;
           "DB_PartManagement".sPosition.sShuttle2.Undrilled.Presence.BW := FALSE;
           "DB_PartManagement".sPosition.sShuttle2.Drilled.Presence.Part := FALSE;
           "DB_PartManagement".sPosition.sShuttle2.Drilled.Presence.BW := FALSE;

           "DB_PartManagement".sPosition.sGripper.Undrilled.Presence.Part := FALSE;
           "DB_PartManagement".sPosition.sGripper.Undrilled.Presence.BW := FALSE;
           "DB_PartManagement".sPosition.sGripper.Drilled.Presence.Part := FALSE;
           "DB_PartManagement".sPosition.sGripper.Drilled.Presence.BW := FALSE;

           "DB_PartManagement".sPosition.sFixture.Undrilled.Presence.Part := FALSE;
           "DB_PartManagement".sPosition.sFixture.Undrilled.Presence.BW := FALSE;
           "DB_PartManagement".sPosition.sFixture.Drilled.Presence.Part := FALSE;
           "DB_PartManagement".sPosition.sFixture.Drilled.Presence.BW := FALSE;

           "DB_WAF".ResetPartPosition := FALSE;
           "DB_WAF".NewTag_2 := FALSE;
       END_IF;
   END_REGION
END_FUNCTION_BLOCK

ORGANIZATION_BLOCK "CyclicInterrupt"   // OB30, SCL, CyclicInterrupt
{ S7_Optimized_Access := 'TRUE' }
// stored: SetENOAutomatically false
   VAR_INPUT
      Initial_Call : Bool;   // Initial call of this OB
      Event_Count : Int;   // Events discarded
   END_VAR
BEGIN
   REGION Description head
       //==================================================================================
       // POSALUX Swiss SA / (C) Copyright 2026
       //----------------------------------------------------------------------------------
       // Title: Hardware interrupt
       // Comment/Function: OB30
       // Author: Fabien WALDT
       // Engineering: TIA Portal v20
       //----------------------------------------------------------------------------------
       // Change log table:
       // Version  | Date     | Expert in charge | Changes applied
       //----------------------------------------------------------------------------------
       // 00.00.01 | 20260501 | WFA              | First released version
       //==================================================================================
   END_REGION

   REGION Machine temperature cooling PID
       "CONT_C_Clim_DB"(COM_RST := "DB_Temperature".sPIDRestart,
                        MAN_ON := FALSE,
                        P_SEL := TRUE,
                        I_SEL := TRUE,
                        INT_HOLD := "DB_Temperature".sPIDHoldI,
                        D_SEL := TRUE,
                        CYCLE := T#1s,
                        SP_INT := "DB_HMISetting".TemperatureCoolingSetpoint,
                        PV_IN := "DB_AnalogInputs".sClimTemperature.sSWRealValue,
                        GAIN := "DB_Temperature".sP,
                        TI := "DB_Temperature".sI,
                        TD := "DB_Temperature".sD,
                        DEADB_W := 0.1,
                        LMN_HLM := 100,
                        LMN_LLM := 0,
                        LMN => "DB_AnalogOutputs".sPropValveClimSetPoint.sSWRealValue);
   END_REGION
END_ORGANIZATION_BLOCK

ORGANIZATION_BLOCK "DiagnosticErrorInterrupt"   // OB82, SCL, DiagnosticErrorInterrupt
{ S7_Optimized_Access := 'TRUE' }
// stored: SetENOAutomatically false
   VAR_INPUT
      IO_State : Word;   // IO state of the HW object
      LADDR : HW_ANY;   // Hardware identifier
      Channel : UInt;   // Channel number
      MultiError : Bool;   // =true if more than one error is present
   END_VAR
BEGIN
   REGION Description head
       //==================================================================================
       // POSALUX Swiss SA / (C) Copyright 2025
       //----------------------------------------------------------------------------------
       // Title: DiagnosticErrorInterrupt
       // Comment/Function: Executes when the CPU detects a diagnostic error,
       //                   or if a diagnostics-capable module recognizes an error
       // Author: Fabien WALDT
       // Engineering: TIA Portal v19
       //----------------------------------------------------------------------------------
       // Change log table:
       // Version  | Date     | Expert in charge | Changes applied
       //----------------------------------------------------------------------------------
       // 00.00.01 | 20250423 | WFA              | First released version
       //==================================================================================
   END_REGION
END_ORGANIZATION_BLOCK

